RoboDK station: InvertedRobot003.rdk

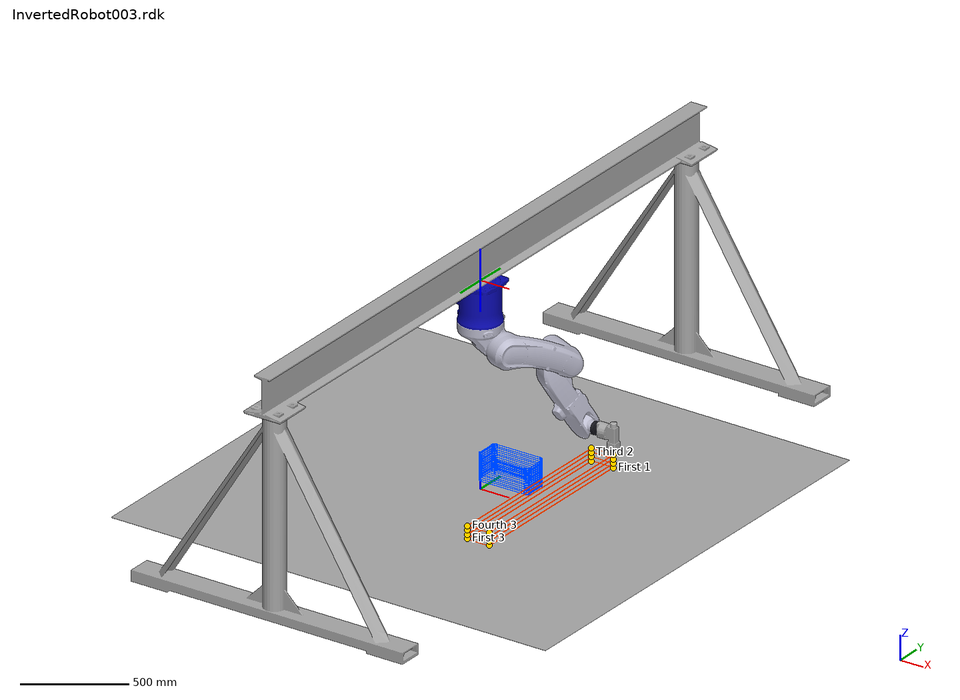
[picture v0: the station drawn from its stored meshes, robots at their saved joint values, targets as dots, program paths as lines]
Station InvertedRobot003 (saved by RoboDK 5.5.4). Poses are relative to the parent item; angles as X-Y-Z fixed-axis rotations.
Station parameters (name, value as stored): TAGS, ['Additive Manufacturing', 'Additive manufacturing']
  - frame Denso 1 at (0, 0, 1066.8) mm, rotated rx -180 ry 0 rz 0 deg
    - robot Denso VS-6577G-B: 6 axes, payload 7 kg, reach 854 mm, repeatability 0.03 mm, weight 36 kg
        modified DH rows (alpha deg, a mm, theta deg, d mm): 0, 0, 0, 335; -90, 75, -90, 0; 0, 365, -90, 0; -90, 90, 0, 405; 90, 0, 0, 0; -90, 0, 0, 80
        joint limits [-170, -100, -119, -190, -120, -360] to [170, 135, 169, 190, 120, 360]; home [0, 0, 90, 0, 0, 0]; saved at [-64.134, 67.115, -35.034, 67.667, 76.602, -29.424]
      - tool nozzle, TCP at (110, 0, 80) mm, rotated rx 0 ry 90 rz 0 deg, size 158.8 x 76.2 x 114.9 mm, geometry from nozzle.STEP
  - frame Ref001 at (0, 0, 0) mm
    - object Part at (0, 0, 0) mm, size 120 x 120 x 160 mm, geometry from part.sld
    - target First 1 (Cartesian target) at (400, 495, 22.23) mm, rotated rx 180 ry 0 rz 180 deg; joints [-64.134, 50.356, -9.939, 69.739, 73.569, -37.461] of Denso VS-6577G-B
    - target First 2 (Cartesian target) at (278, 495, 22.23) mm, rotated rx 180 ry 0 rz 180 deg; joints [-76.592, 55.531, -24.311, 78.477, 83.097, -30.522] of Denso VS-6577G-B
    - target First 3 (Cartesian target) at (278, -500, 22.23) mm, rotated rx 180 ry 0 rz 180 deg; joints [76.721, 17.283, 48.008, -84.366, 77.956, 64.696] of Denso VS-6577G-B
    - target First 4 (Cartesian target) at (400, -500, 22.23) mm, rotated rx 180 ry 0 rz 180 deg; joints [64.359, 49.428, -7.705, -70.29, 73.262, 38.795] of Denso VS-6577G-B
    - target Second 1 (Cartesian target) at (400, 495, 44.45) mm, rotated rx 180 ry 0 rz -180 deg; joints [-64.134, 57.09, -20.57, 68.712, 74.952, -33.676] of Denso VS-6577G-B
    - target Second 2 (Cartesian target) at (278, 495, 44.45) mm, rotated rx 180 ry 0 rz -180 deg; joints [-76.592, 60.643, -31.914, 78.193, 83.601, -28.066] of Denso VS-6577G-B
    - target Second 3 (Cartesian target) at (278, -500, 44.45) mm, rotated rx 180 ry 0 rz -180 deg; joints [76.721, 60.327, -30.755, -78.401, 83.491, 28.91] of Denso VS-6577G-B
    - target Second 4 (Cartesian target) at (400, -500, 44.45) mm, rotated rx 180 ry 0 rz -180 deg; joints [64.359, 56.542, -19.05, -69.151, 74.729, 34.667] of Denso VS-6577G-B
    - target Third 1 (Cartesian target) at (400, 495, 66.67) mm, rotated rx 180 ry 0 rz -180 deg; joints [-64.134, 62.433, -28.479, 68.091, 75.897, -31.211] of Denso VS-6577G-B
    - target Third 2 (Cartesian target) at (278, 495, 66.67) mm, rotated rx 180 ry 0 rz 180 deg; joints [-76.592, 65.197, -38.359, 77.992, 83.991, -26.205] of Denso VS-6577G-B
    - target Third 3 (Cartesian target) at (278, -500, 66.67) mm, rotated rx 180 ry 0 rz 180 deg; joints [76.721, 64.945, -37.316, -78.19, 83.885, 26.996] of Denso VS-6577G-B
    - target Third 4 (Cartesian target) at (400, -500, 66.67) mm, rotated rx 180 ry 0 rz 180 deg; joints [64.359, 62.027, -27.223, -68.489, 75.701, 32.074] of Denso VS-6577G-B
    - target Fourth 1 (Cartesian target) at (400, 495, 88.9) mm, rotated rx 180 ry 0 rz 180 deg; joints [-64.134, 67.115, -35.034, 67.667, 76.602, -29.424] of Denso VS-6577G-B
    - target Fourth 2 (Cartesian target) at (278, 495, 88.9) mm, rotated rx 180 ry 0 rz 180 deg; joints [-76.592, 69.405, -44.036, 77.844, 84.298, -24.761] of Denso VS-6577G-B
    - target Fourth 3 (Cartesian target) at (278, -500, 88.9) mm, rotated rx 180 ry 0 rz 180 deg; joints [76.721, 69.194, -43.068, -78.037, 84.195, 25.517] of Denso VS-6577G-B
    - target Fourth 4 (Cartesian target) at (400, -500, 88.9) mm, rotated rx 180 ry 0 rz 180 deg; joints [64.359, 66.785, -33.922, -68.041, 76.419, 30.216] of Denso VS-6577G-B
  - machining project Print3D settings: C:/Users/silverBlacK/OneDrive - University of Idaho/Research/RoboticsResearch/WallSection.gcode | rotZ(0) | rotX(0)*rotY(0) | rotZ(0)
  - program Print3D (17608 instructions, listed below)
  - frame Frame 4 at (0, 0, 1066.8) mm
    - object GantryAssembly at (0, 0, 0) mm, size 1524 x 3505.2 x 1270 mm, geometry from GantryAssembly.STEP
  - frame GarageFloor at (0, 0, 0) mm
    - object GarageFloor at (0, 0, 0) mm, size 2438.4 x 2438.4 x 2.5 mm, geometry from GarageFloor.STEP
  - program Prog4 (22 instructions, listed below)
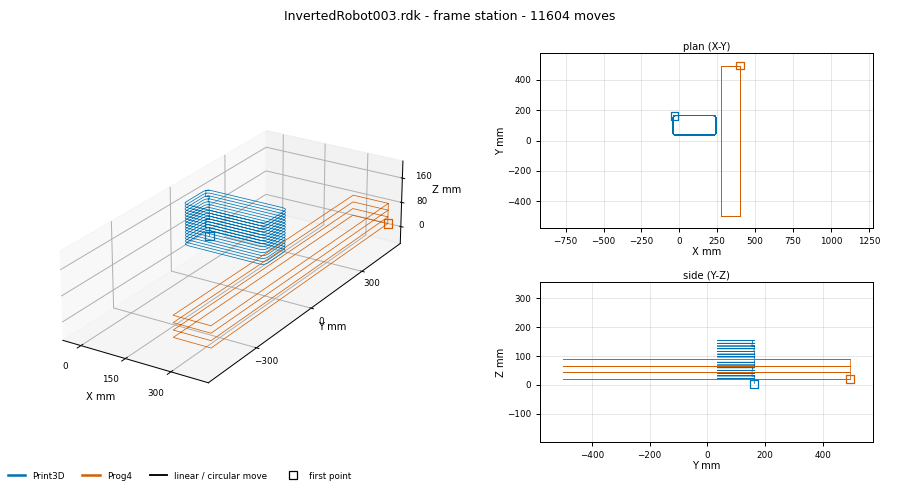
[picture p0: tool path of InvertedRobot003.rdk in frame station, 11604 of 11604 moves have a stored position in this frame; points joined in program order, loops and branches not executed]

--- program Print3D (robot Denso VS-6577G-B) ---
  Smooth(1)
  Call M_RunCode(107)
  Call M_RunCode(104)
  Set speed (83.3 mm/s)
  Set speed (1000.0 mm/s)
  Set Ref.: Ref001
  Set Tool: nozzle
  Show nozzle
  MoveJ 1 to (-31.64, 163.21, 5) mm, rotated rx -180 ry 0 rz 180 deg; joints [-139.581, 53.249, -56.919, 139.523, 87.207, 2.381]
  MoveL 2 to (-31.64, 163.21, 5) mm, rotated rx -180 ry 0 rz 180 deg; joints [-139.581, 53.249, -56.919, 139.523, 87.207, 2.381]
  Call Extruder(-1)
  MoveL 3 to (-31.64, 163.21, 5) mm, rotated rx -180 ry 0 rz 180 deg; joints [-139.581, 53.249, -56.919, 139.523, 87.207, 2.381]
  Call M_RunCode(109)
  Call M_RunCode(82)
  Call Extruder(0.00000)
  Set speed (130.0 mm/s)
  MoveL 4 to (-31.64, 163.21, 22.22) mm, rotated rx 180 ry 0 rz -180 deg; joints [-139.581, 55.977, -61.099, 139.468, 86.103, 3.326]
  Call Extruder(-2.00000)
  Set speed (40.0 mm/s)
  MoveL 5 to (-31.64, 163.21, 22.22) mm, rotated rx 180 ry 0 rz -180 deg; joints [-139.581, 55.977, -61.099, 139.468, 86.103, 3.326]
  Call Extruder(0.00000)
  Set speed (130.0 mm/s)
  MoveL 6 to (-31.64, 163.21, 22.22) mm, rotated rx 180 ry 0 rz -180 deg; joints [-139.581, 55.977, -61.099, 139.468, 86.103, 3.326]
  Call Extruder(2.00000)
  Set speed (40.0 mm/s)
  MoveL 7 to (-31.64, 163.21, 22.22) mm, rotated rx 180 ry 0 rz -180 deg; joints [-139.581, 55.977, -61.099, 139.468, 86.103, 3.326]
  Set speed (30.0 mm/s)
  MoveL 8 to (-31.64, 163.21, 22.22) mm, rotated rx 180 ry 0 rz -180 deg; joints [-139.581, 55.977, -61.099, 139.468, 86.103, 3.326]
  Call Extruder(2.38024)
  MoveL 9 to (-31.93, 163.09, 22.22) mm, rotated rx -180 ry 0 rz 180 deg; joints [-139.645, 55.984, -61.089, 139.532, 86.112, 3.311]
  MoveL 10 to (-31.93, 163.09, 22.22) mm, rotated rx -180 ry 0 rz 180 deg; joints [-139.645, 55.984, -61.089, 139.532, 86.112, 3.311]
  Call Extruder(2.76227)
  MoveL 11 to (-32.22, 162.97, 22.23) mm, rotated rx -180 ry 0 rz -180 deg; joints [-139.709, 55.991, -61.079, 139.597, 86.121, 3.295]
  MoveL 12 to (-32.22, 162.97, 22.23) mm, rotated rx -180 ry 0 rz -180 deg; joints [-139.709, 55.991, -61.079, 139.597, 86.121, 3.295]
  Call Extruder(3.11872)
  MoveL 13 to (-32.49, 162.85, 22.22) mm, rotated rx 180 ry 0 rz 180 deg; joints [-139.768, 55.998, -61.07, 139.657, 86.13, 3.281]
  MoveL 14 to (-32.49, 162.85, 22.22) mm, rotated rx 180 ry 0 rz 180 deg; joints [-139.768, 55.998, -61.07, 139.657, 86.13, 3.281]
  Call Extruder(3.44932)
  MoveL 15 to (-32.74, 162.74, 22.22) mm, rotated rx -180 ry 0 rz 180 deg; joints [-139.823, 56.004, -61.061, 139.713, 86.138, 3.268]
  MoveL 16 to (-32.74, 162.74, 22.22) mm, rotated rx -180 ry 0 rz 180 deg; joints [-139.823, 56.004, -61.061, 139.713, 86.138, 3.268]
  Call Extruder(3.78134)
  MoveL 17 to (-32.99, 162.64, 22.22) mm, rotated rx 180 ry 0 rz -180 deg; joints [-139.878, 56.01, -61.053, 139.769, 86.146, 3.255]
  MoveL 18 to (-32.99, 162.64, 22.22) mm, rotated rx 180 ry 0 rz -180 deg; joints [-139.878, 56.01, -61.053, 139.769, 86.146, 3.255]
  Call Extruder(4.21321)
  MoveL 19 to (-33.29, 162.46, 22.22) mm, rotated rx -180 ry 0 rz 180 deg; joints [-139.953, 56.016, -61.044, 139.844, 86.152, 3.24]
  MoveL 20 to (-33.29, 162.46, 22.22) mm, rotated rx -180 ry 0 rz 180 deg; joints [-139.953, 56.016, -61.044, 139.844, 86.152, 3.24]
  Call Extruder(4.64692)
  MoveL 21 to (-33.6, 162.29, 22.22) mm, rotated rx 180 ry 0 rz 180 deg; joints [-140.028, 56.022, -61.036, 139.92, 86.159, 3.226]
  MoveL 22 to (-33.6, 162.29, 22.22) mm, rotated rx 180 ry 0 rz 180 deg; joints [-140.028, 56.022, -61.036, 139.92, 86.159, 3.226]
  Call Extruder(5.08247)
  MoveL 23 to (-33.9, 162.11, 22.22) mm, rotated rx -180 ry 0 rz 180 deg; joints [-140.103, 56.027, -61.028, 139.995, 86.166, 3.212]
  MoveL 24 to (-33.9, 162.11, 22.22) mm, rotated rx -180 ry 0 rz 180 deg; joints [-140.103, 56.027, -61.028, 139.995, 86.166, 3.212]
  Call Extruder(5.51986)
  MoveL 25 to (-34.21, 161.93, 22.22) mm, rotated rx -180 ry 0 rz -180 deg; joints [-140.178, 56.033, -61.019, 140.071, 86.173, 3.198]
  MoveL 26 to (-34.21, 161.93, 22.22) mm, rotated rx -180 ry 0 rz -180 deg; joints [-140.178, 56.033, -61.019, 140.071, 86.173, 3.198]
  Call Extruder(5.89660)
  MoveL 27 to (-34.45, 161.76, 22.23) mm, rotated rx -180 ry 0 rz 180 deg; joints [-140.244, 56.037, -61.014, 140.137, 86.176, 3.187]
  MoveL 28 to (-34.45, 161.76, 22.23) mm, rotated rx -180 ry 0 rz 180 deg; joints [-140.244, 56.037, -61.014, 140.137, 86.176, 3.187]
  Call Extruder(6.59657)
  MoveL 29 to (-34.9, 161.43, 22.22) mm, rotated rx 180 ry 0 rz -180 deg; joints [-140.366, 56.044, -61.004, 140.261, 86.182, 3.169]
  MoveL 30 to (-34.9, 161.43, 22.22) mm, rotated rx 180 ry 0 rz -180 deg; joints [-140.366, 56.044, -61.004, 140.261, 86.182, 3.169]
  Call Extruder(7.29934)
  MoveL 31 to (-35.35, 161.1, 22.22) mm, rotated rx -180 ry 0 rz -180 deg; joints [-140.489, 56.051, -60.994, 140.384, 86.188, 3.15]
  Call Extruder(9.03811)
  MoveL 32 to (-36.39, 160.19, 22.22) mm, rotated rx -180 ry 0 rz 180 deg; joints [-140.797, 56.062, -60.979, 140.693, 86.192, 3.112]
  Call Extruder(10.77694)
  MoveL 33 to (-37.3, 159.15, 22.22) mm, rotated rx -180 ry 0 rz -180 deg; joints [-141.109, 56.064, -60.975, 141.006, 86.18, 3.087]
  Call Extruder(11.12832)
  MoveL 34 to (-37.47, 158.93, 22.22) mm, rotated rx -180 ry 0 rz -180 deg; joints [-141.172, 56.064, -60.976, 141.069, 86.175, 3.084]
  MoveL 35 to (-37.47, 158.93, 22.22) mm, rotated rx -180 ry 0 rz -180 deg; joints [-141.172, 56.064, -60.976, 141.069, 86.175, 3.084]
  Call Extruder(11.82828)
  MoveL 36 to (-37.8, 158.48, 22.22) mm, rotated rx 180 ry 0 rz 180 deg; joints [-141.298, 56.062, -60.978, 141.195, 86.166, 3.078]
  MoveL 37 to (-37.8, 158.48, 22.22) mm, rotated rx 180 ry 0 rz 180 deg; joints [-141.298, 56.062, -60.978, 141.195, 86.166, 3.078]
  Call Extruder(12.52544)
  MoveL 38 to (-38.12, 158.03, 22.22) mm, rotated rx 180 ry 0 rz 180 deg; joints [-141.424, 56.061, -60.979, 141.321, 86.157, 3.071]
  MoveL 39 to (-38.12, 158.03, 22.22) mm, rotated rx 180 ry 0 rz 180 deg; joints [-141.424, 56.061, -60.979, 141.321, 86.157, 3.071]
  Call Extruder(12.77229)
  MoveL 40 to (-38.22, 157.85, 22.22) mm, rotated rx -180 ry 0 rz 180 deg; joints [-141.468, 56.06, -60.981, 141.365, 86.152, 3.071]
  MoveL 41 to (-38.22, 157.85, 22.22) mm, rotated rx -180 ry 0 rz 180 deg; joints [-141.468, 56.06, -60.981, 141.365, 86.152, 3.071]
  Call Extruder(13.20785)
  MoveL 42 to (-38.4, 157.55, 22.22) mm, rotated rx 180 ry 0 rz -180 deg; joints [-141.547, 56.057, -60.985, 141.443, 86.143, 3.069]
  MoveL 43 to (-38.4, 157.55, 22.22) mm, rotated rx 180 ry 0 rz -180 deg; joints [-141.547, 56.057, -60.985, 141.443, 86.143, 3.069]
  Call Extruder(13.64157)
  MoveL 44 to (-38.57, 157.25, 22.22) mm, rotated rx 180 ry 0 rz 180 deg; joints [-141.625, 56.055, -60.989, 141.522, 86.134, 3.068]
  MoveL 45 to (-38.57, 157.25, 22.22) mm, rotated rx 180 ry 0 rz 180 deg; joints [-141.625, 56.055, -60.989, 141.522, 86.134, 3.068]
  Call Extruder(14.07344)
  MoveL 46 to (-38.75, 156.94, 22.23) mm, rotated rx 180 ry 0 rz 180 deg; joints [-141.704, 56.052, -60.992, 141.6, 86.125, 3.066]
  MoveL 47 to (-38.75, 156.94, 22.23) mm, rotated rx 180 ry 0 rz 180 deg; joints [-141.704, 56.052, -60.992, 141.6, 86.125, 3.066]
  Call Extruder(14.45383)
  MoveL 48 to (-38.89, 156.67, 22.22) mm, rotated rx -180 ry 0 rz -180 deg; joints [-141.773, 56.049, -60.996, 141.669, 86.115, 3.066]
  MoveL 49 to (-38.89, 156.67, 22.22) mm, rotated rx -180 ry 0 rz -180 deg; joints [-141.773, 56.049, -60.996, 141.669, 86.115, 3.066]
  Call Extruder(14.78446)
  MoveL 50 to (-39, 156.42, 22.22) mm, rotated rx -180 ry 0 rz 180 deg; joints [-141.832, 56.046, -61.001, 141.728, 86.106, 3.067]
  MoveL 51 to (-39, 156.42, 22.22) mm, rotated rx -180 ry 0 rz 180 deg; joints [-141.832, 56.046, -61.001, 141.728, 86.106, 3.067]
  Call Extruder(15.11366)
  MoveL 52 to (-39.1, 156.17, 22.22) mm, rotated rx -180 ry 0 rz -180 deg; joints [-141.891, 56.042, -61.006, 141.787, 86.096, 3.068]
  MoveL 53 to (-39.1, 156.17, 22.22) mm, rotated rx -180 ry 0 rz -180 deg; joints [-141.891, 56.042, -61.006, 141.787, 86.096, 3.068]
  Call Extruder(15.49565)
  MoveL 54 to (-39.22, 155.87, 22.23) mm, rotated rx -180 ry 0 rz 180 deg; joints [-141.96, 56.038, -61.012, 141.855, 86.084, 3.07]
  MoveL 55 to (-39.22, 155.87, 22.23) mm, rotated rx -180 ry 0 rz 180 deg; joints [-141.96, 56.038, -61.012, 141.855, 86.084, 3.07]
  Call Extruder(15.87585)
  MoveL 56 to (-39.35, 155.58, 22.23) mm, rotated rx 180 ry 0 rz 180 deg; joints [-142.029, 56.034, -61.018, 141.924, 86.073, 3.071]
  MoveL 57 to (-39.35, 155.58, 22.23) mm, rotated rx 180 ry 0 rz 180 deg; joints [-142.029, 56.034, -61.018, 141.924, 86.073, 3.071]
  Call Extruder(16.18353)
  MoveL 58 to (-39.44, 155.34, 22.22) mm, rotated rx 180 ry 0 rz 180 deg; joints [-142.085, 56.03, -61.024, 141.979, 86.063, 3.073]
  MoveL 59 to (-39.44, 155.34, 22.22) mm, rotated rx 180 ry 0 rz 180 deg; joints [-142.085, 56.03, -61.024, 141.979, 86.063, 3.073]
  Call Extruder(16.41988)
  MoveL 60 to (-39.5, 155.15, 22.22) mm, rotated rx -180 ry 0 rz 180 deg; joints [-142.127, 56.027, -61.028, 142.021, 86.054, 3.075]
  MoveL 61 to (-39.5, 155.15, 22.22) mm, rotated rx -180 ry 0 rz 180 deg; joints [-142.127, 56.027, -61.028, 142.021, 86.054, 3.075]
  Call Extruder(16.65518)
  MoveL 62 to (-39.56, 154.97, 22.22) mm, rotated rx -180 ry 0 rz 180 deg; joints [-142.169, 56.024, -61.033, 142.063, 86.045, 3.077]
  MoveL 63 to (-39.56, 154.97, 22.22) mm, rotated rx -180 ry 0 rz 180 deg; joints [-142.169, 56.024, -61.033, 142.063, 86.045, 3.077]
  Call Extruder(16.88943)
  MoveL 64 to (-39.62, 154.78, 22.22) mm, rotated rx 180 ry 0 rz 180 deg; joints [-142.212, 56.02, -61.038, 142.105, 86.037, 3.079]
  MoveL 65 to (-39.62, 154.78, 22.22) mm, rotated rx 180 ry 0 rz 180 deg; joints [-142.212, 56.02, -61.038, 142.105, 86.037, 3.079]
  Call Extruder(17.12262)
  MoveL 66 to (-39.68, 154.59, 22.22) mm, rotated rx -180 ry 0 rz -180 deg; joints [-142.254, 56.017, -61.042, 142.147, 86.028, 3.081]
  MoveL 67 to (-39.68, 154.59, 22.22) mm, rotated rx -180 ry 0 rz -180 deg; joints [-142.254, 56.017, -61.042, 142.147, 86.028, 3.081]
  Call Extruder(17.37548)
  MoveL 68 to (-39.75, 154.38, 22.22) mm, rotated rx -180 ry 0 rz 180 deg; joints [-142.3, 56.013, -61.048, 142.193, 86.019, 3.084]
  MoveL 69 to (-39.75, 154.38, 22.22) mm, rotated rx -180 ry 0 rz 180 deg; joints [-142.3, 56.013, -61.048, 142.193, 86.019, 3.084]
  Call Extruder(17.64775)
  MoveL 70 to (-39.81, 154.16, 22.22) mm, rotated rx 180 ry 0 rz 180 deg; joints [-142.35, 56.009, -61.053, 142.242, 86.008, 3.086]
  MoveL 71 to (-39.81, 154.16, 22.22) mm, rotated rx 180 ry 0 rz 180 deg; joints [-142.35, 56.009, -61.053, 142.242, 86.008, 3.086]
  Call Extruder(17.91868)
  MoveL 72 to (-39.88, 153.94, 22.22) mm, rotated rx 180 ry 0 rz -180 deg; joints [-142.399, 56.005, -61.059, 142.291, 85.998, 3.089]
  MoveL 73 to (-39.88, 153.94, 22.22) mm, rotated rx 180 ry 0 rz -180 deg; joints [-142.399, 56.005, -61.059, 142.291, 85.998, 3.089]
  Call Extruder(18.18828)
  MoveL 74 to (-39.95, 153.71, 22.23) mm, rotated rx -180 ry 0 rz -180 deg; joints [-142.449, 56.001, -61.065, 142.34, 85.987, 3.091]
  MoveL 75 to (-39.95, 153.71, 22.23) mm, rotated rx -180 ry 0 rz -180 deg; joints [-142.449, 56.001, -61.065, 142.34, 85.987, 3.091]
  Call Extruder(18.45654)
  MoveL 76 to (-40.02, 153.49, 22.22) mm, rotated rx -180 ry 0 rz -180 deg; joints [-142.498, 55.997, -61.071, 142.39, 85.977, 3.094]
  MoveL 77 to (-40.02, 153.49, 22.22) mm, rotated rx -180 ry 0 rz -180 deg; joints [-142.498, 55.997, -61.071, 142.39, 85.977, 3.094]
  Call Extruder(18.69554)
  MoveL 78 to (-40.06, 153.28, 22.22) mm, rotated rx -180 ry 0 rz 180 deg; joints [-142.541, 55.993, -61.077, 142.432, 85.966, 3.097]
  MoveL 79 to (-40.06, 153.28, 22.22) mm, rotated rx -180 ry 0 rz 180 deg; joints [-142.541, 55.993, -61.077, 142.432, 85.966, 3.097]
  Call Extruder(18.93348)
  MoveL 80 to (-40.11, 153.08, 22.22) mm, rotated rx 180 ry 0 rz 180 deg; joints [-142.584, 55.988, -61.083, 142.475, 85.955, 3.101]
  MoveL 81 to (-40.11, 153.08, 22.22) mm, rotated rx 180 ry 0 rz 180 deg; joints [-142.584, 55.988, -61.083, 142.475, 85.955, 3.101]
  Call Extruder(19.17035)
  MoveL 82 to (-40.15, 152.88, 22.22) mm, rotated rx -180 ry 0 rz 180 deg; joints [-142.627, 55.984, -61.089, 142.517, 85.945, 3.104]
  MoveL 83 to (-40.15, 152.88, 22.22) mm, rotated rx -180 ry 0 rz 180 deg; joints [-142.627, 55.984, -61.089, 142.517, 85.945, 3.104]
  Call Extruder(19.40615)
  MoveL 84 to (-40.2, 152.67, 22.22) mm, rotated rx -180 ry 0 rz 180 deg; joints [-142.671, 55.979, -61.096, 142.56, 85.934, 3.108]
  MoveL 85 to (-40.2, 152.67, 22.22) mm, rotated rx -180 ry 0 rz 180 deg; joints [-142.671, 55.979, -61.096, 142.56, 85.934, 3.108]
  Call Extruder(19.66605)
  MoveL 86 to (-40.24, 152.44, 22.22) mm, rotated rx 180 ry 0 rz 180 deg; joints [-142.718, 55.974, -61.103, 142.607, 85.922, 3.112]
  MoveL 87 to (-40.24, 152.44, 22.22) mm, rotated rx 180 ry 0 rz 180 deg; joints [-142.718, 55.974, -61.103, 142.607, 85.922, 3.112]
  Call Extruder(19.94972)
  MoveL 88 to (-40.29, 152.2, 22.23) mm, rotated rx -180 ry 0 rz -180 deg; joints [-142.77, 55.969, -61.11, 142.659, 85.908, 3.116]
  MoveL 89 to (-40.29, 152.2, 22.23) mm, rotated rx -180 ry 0 rz -180 deg; joints [-142.77, 55.969, -61.11, 142.659, 85.908, 3.116]
  Call Extruder(20.23193)
  MoveL 90 to (-40.34, 151.95, 22.22) mm, rotated rx -180 ry 0 rz -180 deg; joints [-142.822, 55.963, -61.118, 142.71, 85.895, 3.12]
  MoveL 91 to (-40.34, 151.95, 22.22) mm, rotated rx -180 ry 0 rz -180 deg; joints [-142.822, 55.963, -61.118, 142.71, 85.895, 3.12]
  Call Extruder(20.51271)
  MoveL 92 to (-40.39, 151.7, 22.22) mm, rotated rx 180 ry 0 rz 180 deg; joints [-142.874, 55.958, -61.126, 142.762, 85.882, 3.125]
  MoveL 93 to (-40.39, 151.7, 22.22) mm, rotated rx 180 ry 0 rz 180 deg; joints [-142.874, 55.958, -61.126, 142.762, 85.882, 3.125]
  Call Extruder(20.79205)
  MoveL 94 to (-40.44, 151.45, 22.23) mm, rotated rx 180 ry 0 rz 180 deg; joints [-142.926, 55.952, -61.133, 142.813, 85.868, 3.129]
  MoveL 95 to (-40.44, 151.45, 22.23) mm, rotated rx 180 ry 0 rz 180 deg; joints [-142.926, 55.952, -61.133, 142.813, 85.868, 3.129]
  Call Extruder(21.06994)
  MoveL 96 to (-40.49, 151.2, 22.23) mm, rotated rx -180 ry 0 rz 180 deg; joints [-142.978, 55.947, -61.141, 142.865, 85.855, 3.133]
  MoveL 97 to (-40.49, 151.2, 22.23) mm, rotated rx -180 ry 0 rz 180 deg; joints [-142.978, 55.947, -61.141, 142.865, 85.855, 3.133]
  Call Extruder(21.34639)
  MoveL 98 to (-40.54, 150.95, 22.23) mm, rotated rx 180 ry 0 rz 180 deg; joints [-143.031, 55.941, -61.149, 142.917, 85.842, 3.137]
  MoveL 99 to (-40.54, 150.95, 22.23) mm, rotated rx 180 ry 0 rz 180 deg; joints [-143.031, 55.941, -61.149, 142.917, 85.842, 3.137]
  Call Extruder(21.65140)
  MoveL 100 to (-40.59, 150.67, 22.22) mm, rotated rx -180 ry 0 rz -180 deg; joints [-143.088, 55.935, -61.158, 142.973, 85.826, 3.142]
  MoveL 101 to (-40.59, 150.67, 22.22) mm, rotated rx -180 ry 0 rz -180 deg; joints [-143.088, 55.935, -61.158, 142.973, 85.826, 3.142]
  Call Extruder(21.98479)
  MoveL 102 to (-40.64, 150.37, 22.22) mm, rotated rx 180 ry 0 rz -180 deg; joints [-143.15, 55.928, -61.168, 143.035, 85.809, 3.148]
  MoveL 103 to (-40.64, 150.37, 22.22) mm, rotated rx 180 ry 0 rz -180 deg; joints [-143.15, 55.928, -61.168, 143.035, 85.809, 3.148]
  Call Extruder(22.31647)
  MoveL 104 to (-40.69, 150.06, 22.22) mm, rotated rx 180 ry 0 rz 180 deg; joints [-143.213, 55.921, -61.178, 143.097, 85.792, 3.154]
  MoveL 105 to (-40.69, 150.06, 22.22) mm, rotated rx 180 ry 0 rz 180 deg; joints [-143.213, 55.921, -61.178, 143.097, 85.792, 3.154]
  Call Extruder(22.64643)
  MoveL 106 to (-40.74, 149.76, 22.22) mm, rotated rx -180 ry 0 rz -180 deg; joints [-143.276, 55.913, -61.188, 143.159, 85.775, 3.16]
  MoveL 107 to (-40.74, 149.76, 22.22) mm, rotated rx -180 ry 0 rz -180 deg; joints [-143.276, 55.913, -61.188, 143.159, 85.775, 3.16]
  Call Extruder(22.97467)
  MoveL 108 to (-40.78, 149.45, 22.22) mm, rotated rx 180 ry 0 rz 180 deg; joints [-143.338, 55.906, -61.198, 143.221, 85.758, 3.165]
  MoveL 109 to (-40.78, 149.45, 22.22) mm, rotated rx 180 ry 0 rz 180 deg; joints [-143.338, 55.906, -61.198, 143.221, 85.758, 3.165]
  Call Extruder(23.30119)
  MoveL 110 to (-40.83, 149.14, 22.22) mm, rotated rx -180 ry 0 rz 180 deg; joints [-143.401, 55.899, -61.207, 143.283, 85.74, 3.171]
  MoveL 111 to (-40.83, 149.14, 22.22) mm, rotated rx -180 ry 0 rz 180 deg; joints [-143.401, 55.899, -61.207, 143.283, 85.74, 3.171]
  Call Extruder(23.66827)
  MoveL 112 to (-40.88, 148.8, 22.22) mm, rotated rx -180 ry 0 rz 180 deg; joints [-143.471, 55.891, -61.219, 143.353, 85.72, 3.178]
  MoveL 113 to (-40.88, 148.8, 22.22) mm, rotated rx -180 ry 0 rz 180 deg; joints [-143.471, 55.891, -61.219, 143.353, 85.72, 3.178]
  Call Extruder(24.07571)
  MoveL 114 to (-40.93, 148.41, 22.22) mm, rotated rx 180 ry 0 rz 180 deg; joints [-143.549, 55.881, -61.232, 143.429, 85.698, 3.186]
  MoveL 115 to (-40.93, 148.41, 22.22) mm, rotated rx 180 ry 0 rz 180 deg; joints [-143.549, 55.881, -61.232, 143.429, 85.698, 3.186]
  Call Extruder(24.48110)
  MoveL 116 to (-40.97, 148.02, 22.22) mm, rotated rx -180 ry 0 rz -180 deg; joints [-143.627, 55.871, -61.246, 143.506, 85.675, 3.193]
  MoveL 117 to (-40.97, 148.02, 22.22) mm, rotated rx -180 ry 0 rz -180 deg; joints [-143.627, 55.871, -61.246, 143.506, 85.675, 3.193]
  Call Extruder(24.88445)
  MoveL 118 to (-41.02, 147.63, 22.22) mm, rotated rx -180 ry 0 rz -180 deg; joints [-143.705, 55.861, -61.259, 143.583, 85.652, 3.201]
  MoveL 119 to (-41.02, 147.63, 22.22) mm, rotated rx -180 ry 0 rz -180 deg; joints [-143.705, 55.861, -61.259, 143.583, 85.652, 3.201]
  Call Extruder(25.28574)
  MoveL 120 to (-41.06, 147.25, 22.22) mm, rotated rx 180 ry 0 rz 180 deg; joints [-143.783, 55.852, -61.272, 143.66, 85.629, 3.209]
  MoveL 121 to (-41.06, 147.25, 22.22) mm, rotated rx 180 ry 0 rz 180 deg; joints [-143.783, 55.852, -61.272, 143.66, 85.629, 3.209]
  Call Extruder(25.89062)
  MoveL 122 to (-41.11, 146.66, 22.22) mm, rotated rx 180 ry 0 rz -180 deg; joints [-143.899, 55.836, -61.293, 143.775, 85.593, 3.222]
  MoveL 123 to (-41.11, 146.66, 22.22) mm, rotated rx 180 ry 0 rz -180 deg; joints [-143.899, 55.836, -61.293, 143.775, 85.593, 3.222]
  Call Extruder(26.49235)
  MoveL 124 to (-41.16, 146.07, 22.22) mm, rotated rx -180 ry 0 rz -180 deg; joints [-144.015, 55.82, -61.315, 143.889, 85.557, 3.235]
  MoveL 125 to (-41.16, 146.07, 22.22) mm, rotated rx -180 ry 0 rz -180 deg; joints [-144.015, 55.82, -61.315, 143.889, 85.557, 3.235]
  Call Extruder(27.09093)
  MoveL 126 to (-41.2, 145.48, 22.22) mm, rotated rx 180 ry 0 rz 180 deg; joints [-144.131, 55.805, -61.336, 144.004, 85.52, 3.247]
  MoveL 127 to (-41.2, 145.48, 22.22) mm, rotated rx 180 ry 0 rz 180 deg; joints [-144.131, 55.805, -61.336, 144.004, 85.52, 3.247]
  Call Extruder(28.26271)
  MoveL 128 to (-41.25, 144.32, 22.22) mm, rotated rx 180 ry 0 rz 180 deg; joints [-144.355, 55.772, -61.379, 144.225, 85.446, 3.274]
  MoveL 129 to (-41.25, 144.32, 22.22) mm, rotated rx 180 ry 0 rz 180 deg; joints [-144.355, 55.772, -61.379, 144.225, 85.446, 3.274]
  Call Extruder(29.72057)
  MoveL 130 to (-41.29, 142.86, 22.22) mm, rotated rx -180 ry 0 rz 180 deg; joints [-144.635, 55.731, -61.434, 144.501, 85.351, 3.308]
  Call Extruder(115.61408)
  MoveL 131 to (-41.29, 57.14, 22.22) mm, rotated rx -180 ry 0 rz 180 deg; joints [-164.153, 53.6, -63.687, 163.917, 80.3, 2.781]
  Call Extruder(116.48916)
  MoveL 132 to (-41.27, 56.26, 22.22) mm, rotated rx -180 ry 0 rz 180 deg; joints [-164.382, 53.584, -63.7, 164.148, 80.261, 2.75]
  MoveL 133 to (-41.27, 56.26, 22.22) mm, rotated rx -180 ry 0 rz 180 deg; joints [-164.382, 53.584, -63.7, 164.148, 80.261, 2.75]
  Call Extruder(117.66094)
  MoveL 134 to (-41.22, 55.1, 22.22) mm, rotated rx 180 ry 0 rz 180 deg; joints [-164.686, 53.562, -63.719, 164.454, 80.207, 2.709]
  MoveL 135 to (-41.22, 55.1, 22.22) mm, rotated rx 180 ry 0 rz 180 deg; joints [-164.686, 53.562, -63.719, 164.454, 80.207, 2.709]
  Call Extruder(118.54904)
  MoveL 136 to (-41.18, 54.23, 22.23) mm, rotated rx 180 ry 0 rz -180 deg; joints [-164.915, 53.545, -63.733, 164.685, 80.166, 2.678]
  MoveL 137 to (-41.18, 54.23, 22.23) mm, rotated rx 180 ry 0 rz -180 deg; joints [-164.915, 53.545, -63.733, 164.685, 80.166, 2.678]
  Call Extruder(119.15077)
  MoveL 138 to (-41.13, 53.64, 22.22) mm, rotated rx 180 ry 0 rz 180 deg; joints [-165.068, 53.532, -63.743, 164.839, 80.137, 2.657]
  MoveL 139 to (-41.13, 53.64, 22.22) mm, rotated rx 180 ry 0 rz 180 deg; joints [-165.068, 53.532, -63.743, 164.839, 80.137, 2.657]
  Call Extruder(119.75565)
  MoveL 140 to (-41.09, 53.05, 22.22) mm, rotated rx -180 ry 0 rz 180 deg; joints [-165.222, 53.52, -63.754, 164.994, 80.109, 2.637]
  MoveL 141 to (-41.09, 53.05, 22.22) mm, rotated rx -180 ry 0 rz 180 deg; joints [-165.222, 53.52, -63.754, 164.994, 80.109, 2.637]
  Call Extruder(120.26021)
  MoveL 142 to (-41.04, 52.56, 22.22) mm, rotated rx -180 ry 0 rz -180 deg; joints [-165.349, 53.51, -63.762, 165.121, 80.084, 2.619]
  MoveL 143 to (-41.04, 52.56, 22.22) mm, rotated rx -180 ry 0 rz -180 deg; joints [-165.349, 53.51, -63.762, 165.121, 80.084, 2.619]
  Call Extruder(120.66355)
  MoveL 144 to (-40.99, 52.17, 22.22) mm, rotated rx -180 ry 0 rz 180 deg; joints [-165.449, 53.501, -63.77, 165.223, 80.064, 2.606]
  MoveL 145 to (-40.99, 52.17, 22.22) mm, rotated rx -180 ry 0 rz 180 deg; joints [-165.449, 53.501, -63.77, 165.223, 80.064, 2.606]
  Call Extruder(121.06894)
  MoveL 146 to (-40.95, 51.78, 22.22) mm, rotated rx -180 ry 0 rz 180 deg; joints [-165.549, 53.492, -63.777, 165.323, 80.044, 2.593]
  MoveL 147 to (-40.95, 51.78, 22.22) mm, rotated rx -180 ry 0 rz 180 deg; joints [-165.549, 53.492, -63.777, 165.323, 80.044, 2.593]
  Call Extruder(121.47639)
  MoveL 148 to (-40.9, 51.4, 22.22) mm, rotated rx 180 ry 0 rz 180 deg; joints [-165.65, 53.483, -63.784, 165.425, 80.024, 2.579]
  MoveL 149 to (-40.9, 51.4, 22.22) mm, rotated rx 180 ry 0 rz 180 deg; joints [-165.65, 53.483, -63.784, 165.425, 80.024, 2.579]
  Call Extruder(121.88588)
  MoveL 150 to (-40.86, 51.01, 22.23) mm, rotated rx 180 ry 0 rz -180 deg; joints [-165.751, 53.474, -63.791, 165.526, 80.004, 2.566]
  MoveL 151 to (-40.86, 51.01, 22.23) mm, rotated rx 180 ry 0 rz -180 deg; joints [-165.751, 53.474, -63.791, 165.526, 80.004, 2.566]
  Call Extruder(122.21240)
  MoveL 152 to (-40.81, 50.7, 22.22) mm, rotated rx 180 ry 0 rz -180 deg; joints [-165.829, 53.467, -63.798, 165.605, 79.987, 2.555]
  MoveL 153 to (-40.81, 50.7, 22.22) mm, rotated rx 180 ry 0 rz -180 deg; joints [-165.829, 53.467, -63.798, 165.605, 79.987, 2.555]
  Call Extruder(122.54064)
  MoveL 154 to (-40.76, 50.4, 22.22) mm, rotated rx -180 ry 0 rz -180 deg; joints [-165.908, 53.459, -63.804, 165.685, 79.97, 2.545]
  MoveL 155 to (-40.76, 50.4, 22.22) mm, rotated rx -180 ry 0 rz -180 deg; joints [-165.908, 53.459, -63.804, 165.685, 79.97, 2.545]
  Call Extruder(122.87060)
  MoveL 156 to (-40.71, 50.09, 22.22) mm, rotated rx 180 ry 0 rz 180 deg; joints [-165.987, 53.451, -63.81, 165.764, 79.953, 2.534]
  MoveL 157 to (-40.71, 50.09, 22.22) mm, rotated rx 180 ry 0 rz 180 deg; joints [-165.987, 53.451, -63.81, 165.764, 79.953, 2.534]
  Call Extruder(123.20228)
  MoveL 158 to (-40.66, 49.79, 22.22) mm, rotated rx -180 ry 0 rz -180 deg; joints [-166.066, 53.444, -63.816, 165.844, 79.936, 2.524]
  MoveL 159 to (-40.66, 49.79, 22.22) mm, rotated rx -180 ry 0 rz -180 deg; joints [-166.066, 53.444, -63.816, 165.844, 79.936, 2.524]
  Call Extruder(123.53568)
  MoveL 160 to (-40.61, 49.48, 22.22) mm, rotated rx -180 ry 0 rz 180 deg; joints [-166.145, 53.436, -63.823, 165.923, 79.919, 2.513]
  MoveL 161 to (-40.61, 49.48, 22.22) mm, rotated rx -180 ry 0 rz 180 deg; joints [-166.145, 53.436, -63.823, 165.923, 79.919, 2.513]
  Call Extruder(123.87079)
  MoveL 162 to (-40.57, 49.17, 22.22) mm, rotated rx -180 ry 0 rz -180 deg; joints [-166.224, 53.429, -63.829, 166.003, 79.902, 2.503]
  MoveL 163 to (-40.57, 49.17, 22.22) mm, rotated rx -180 ry 0 rz -180 deg; joints [-166.224, 53.429, -63.829, 166.003, 79.902, 2.503]
  Call Extruder(124.14680)
  MoveL 164 to (-40.52, 48.93, 22.22) mm, rotated rx 180 ry 0 rz -180 deg; joints [-166.288, 53.422, -63.834, 166.067, 79.888, 2.494]
  MoveL 165 to (-40.52, 48.93, 22.22) mm, rotated rx 180 ry 0 rz -180 deg; joints [-166.288, 53.422, -63.834, 166.067, 79.888, 2.494]
  Call Extruder(124.42424)
  MoveL 166 to (-40.47, 48.68, 22.22) mm, rotated rx -180 ry 0 rz 180 deg; joints [-166.352, 53.415, -63.84, 166.131, 79.873, 2.486]
  MoveL 167 to (-40.47, 48.68, 22.22) mm, rotated rx -180 ry 0 rz 180 deg; joints [-166.352, 53.415, -63.84, 166.131, 79.873, 2.486]
  Call Extruder(124.70312)
  MoveL 168 to (-40.42, 48.43, 22.22) mm, rotated rx -180 ry 0 rz -180 deg; joints [-166.416, 53.409, -63.845, 166.196, 79.859, 2.477]
  MoveL 169 to (-40.42, 48.43, 22.22) mm, rotated rx -180 ry 0 rz -180 deg; joints [-166.416, 53.409, -63.845, 166.196, 79.859, 2.477]
  Call Extruder(124.98344)
  MoveL 170 to (-40.37, 48.18, 22.22) mm, rotated rx -180 ry 0 rz -180 deg; joints [-166.479, 53.402, -63.851, 166.26, 79.844, 2.469]
  MoveL 171 to (-40.37, 48.18, 22.22) mm, rotated rx -180 ry 0 rz -180 deg; joints [-166.479, 53.402, -63.851, 166.26, 79.844, 2.469]
  Call Extruder(125.26519)
  MoveL 172 to (-40.32, 47.93, 22.22) mm, rotated rx 180 ry 0 rz -180 deg; joints [-166.544, 53.395, -63.856, 166.325, 79.829, 2.46]
  MoveL 173 to (-40.32, 47.93, 22.22) mm, rotated rx 180 ry 0 rz -180 deg; joints [-166.544, 53.395, -63.856, 166.325, 79.829, 2.46]
  Call Extruder(125.54838)
  MoveL 174 to (-40.27, 47.68, 22.23) mm, rotated rx -180 ry 0 rz 180 deg; joints [-166.608, 53.388, -63.861, 166.389, 79.815, 2.452]
  MoveL 175 to (-40.27, 47.68, 22.23) mm, rotated rx -180 ry 0 rz 180 deg; joints [-166.608, 53.388, -63.861, 166.389, 79.815, 2.452]
  Call Extruder(125.76334)
  MoveL 176 to (-40.23, 47.49, 22.22) mm, rotated rx 180 ry 0 rz -180 deg; joints [-166.656, 53.383, -63.865, 166.438, 79.804, 2.445]
  MoveL 177 to (-40.23, 47.49, 22.22) mm, rotated rx 180 ry 0 rz -180 deg; joints [-166.656, 53.383, -63.865, 166.438, 79.804, 2.445]
  Call Extruder(125.95387)
  MoveL 178 to (-40.2, 47.33, 22.22) mm, rotated rx -180 ry 0 rz -180 deg; joints [-166.699, 53.379, -63.869, 166.481, 79.794, 2.439]
  MoveL 179 to (-40.2, 47.33, 22.22) mm, rotated rx -180 ry 0 rz -180 deg; joints [-166.699, 53.379, -63.869, 166.481, 79.794, 2.439]
  Call Extruder(126.19017)
  MoveL 180 to (-40.15, 47.12, 22.22) mm, rotated rx -180 ry 0 rz 180 deg; joints [-166.751, 53.373, -63.874, 166.534, 79.782, 2.432]
  MoveL 181 to (-40.15, 47.12, 22.22) mm, rotated rx -180 ry 0 rz 180 deg; joints [-166.751, 53.373, -63.874, 166.534, 79.782, 2.432]
  Call Extruder(126.42754)
  MoveL 182 to (-40.11, 46.92, 22.22) mm, rotated rx -180 ry 0 rz -180 deg; joints [-166.804, 53.367, -63.878, 166.587, 79.77, 2.425]
  MoveL 183 to (-40.11, 46.92, 22.22) mm, rotated rx -180 ry 0 rz -180 deg; joints [-166.804, 53.367, -63.878, 166.587, 79.77, 2.425]
  Call Extruder(126.66598)
  MoveL 184 to (-40.06, 46.72, 22.23) mm, rotated rx 180 ry 0 rz -180 deg; joints [-166.857, 53.362, -63.883, 166.64, 79.758, 2.418]
  MoveL 185 to (-40.06, 46.72, 22.23) mm, rotated rx 180 ry 0 rz -180 deg; joints [-166.857, 53.362, -63.883, 166.64, 79.758, 2.418]
  Call Extruder(126.90549)
  MoveL 186 to (-40.02, 46.51, 22.22) mm, rotated rx -180 ry 0 rz 180 deg; joints [-166.909, 53.356, -63.887, 166.693, 79.745, 2.411]
  MoveL 187 to (-40.02, 46.51, 22.22) mm, rotated rx -180 ry 0 rz 180 deg; joints [-166.909, 53.356, -63.887, 166.693, 79.745, 2.411]
  Call Extruder(127.17442)
  MoveL 188 to (-39.95, 46.29, 22.22) mm, rotated rx -180 ry 0 rz -180 deg; joints [-166.966, 53.349, -63.893, 166.75, 79.73, 2.404]
  MoveL 189 to (-39.95, 46.29, 22.22) mm, rotated rx -180 ry 0 rz -180 deg; joints [-166.966, 53.349, -63.893, 166.75, 79.73, 2.404]
  Call Extruder(127.44468)
  MoveL 190 to (-39.88, 46.06, 22.22) mm, rotated rx 180 ry 0 rz 180 deg; joints [-167.022, 53.341, -63.899, 166.807, 79.715, 2.397]
  MoveL 191 to (-39.88, 46.06, 22.22) mm, rotated rx 180 ry 0 rz 180 deg; joints [-167.022, 53.341, -63.899, 166.807, 79.715, 2.397]
  Call Extruder(127.71628)
  MoveL 192 to (-39.82, 45.84, 22.22) mm, rotated rx 180 ry 0 rz -180 deg; joints [-167.079, 53.334, -63.905, 166.864, 79.7, 2.39]
  MoveL 193 to (-39.82, 45.84, 22.22) mm, rotated rx 180 ry 0 rz -180 deg; joints [-167.079, 53.334, -63.905, 166.864, 79.7, 2.39]
  Call Extruder(127.98921)
  MoveL 194 to (-39.75, 45.62, 22.22) mm, rotated rx 180 ry 0 rz -180 deg; joints [-167.136, 53.327, -63.911, 166.921, 79.684, 2.382]
  MoveL 195 to (-39.75, 45.62, 22.22) mm, rotated rx 180 ry 0 rz -180 deg; joints [-167.136, 53.327, -63.911, 166.921, 79.684, 2.382]
  Call Extruder(128.24265)
  MoveL 196 to (-39.68, 45.41, 22.22) mm, rotated rx -180 ry 0 rz 180 deg; joints [-167.188, 53.32, -63.916, 166.973, 79.67, 2.376]
  MoveL 197 to (-39.68, 45.41, 22.22) mm, rotated rx -180 ry 0 rz 180 deg; joints [-167.188, 53.32, -63.916, 166.973, 79.67, 2.376]
  Call Extruder(128.47637)
  MoveL 198 to (-39.62, 45.22, 22.22) mm, rotated rx 180 ry 0 rz 180 deg; joints [-167.235, 53.313, -63.922, 167.021, 79.657, 2.37]
  MoveL 199 to (-39.62, 45.22, 22.22) mm, rotated rx 180 ry 0 rz 180 deg; joints [-167.235, 53.313, -63.922, 167.021, 79.657, 2.37]
  Call Extruder(128.71114)
  MoveL 200 to (-39.56, 45.03, 22.22) mm, rotated rx 180 ry 0 rz 180 deg; joints [-167.283, 53.307, -63.927, 167.069, 79.644, 2.364]
  MoveL 201 to (-39.56, 45.03, 22.22) mm, rotated rx 180 ry 0 rz 180 deg; joints [-167.283, 53.307, -63.927, 167.069, 79.644, 2.364]
  Call Extruder(128.94697)
  MoveL 202 to (-39.5, 44.85, 22.22) mm, rotated rx -180 ry 0 rz 180 deg; joints [-167.331, 53.3, -63.932, 167.117, 79.63, 2.357]
  MoveL 203 to (-39.5, 44.85, 22.22) mm, rotated rx -180 ry 0 rz 180 deg; joints [-167.331, 53.3, -63.932, 167.117, 79.63, 2.357]
  Call Extruder(129.18384)
  MoveL 204 to (-39.44, 44.66, 22.22) mm, rotated rx -180 ry 0 rz 180 deg; joints [-167.379, 53.294, -63.937, 167.165, 79.617, 2.351]
  MoveL 205 to (-39.44, 44.66, 22.22) mm, rotated rx -180 ry 0 rz 180 deg; joints [-167.379, 53.294, -63.937, 167.165, 79.617, 2.351]
  Call Extruder(129.49225)
  MoveL 206 to (-39.35, 44.42, 22.23) mm, rotated rx -180 ry 0 rz 180 deg; joints [-167.439, 53.285, -63.944, 167.226, 79.599, 2.344]
  MoveL 207 to (-39.35, 44.42, 22.23) mm, rotated rx -180 ry 0 rz 180 deg; joints [-167.439, 53.285, -63.944, 167.226, 79.599, 2.344]
  Call Extruder(129.87335)
  MoveL 208 to (-39.22, 44.12, 22.22) mm, rotated rx 180 ry 0 rz 180 deg; joints [-167.512, 53.274, -63.953, 167.299, 79.576, 2.335]
  MoveL 209 to (-39.22, 44.12, 22.22) mm, rotated rx 180 ry 0 rz 180 deg; joints [-167.512, 53.274, -63.953, 167.299, 79.576, 2.335]
  Call Extruder(130.25623)
  MoveL 210 to (-39.11, 43.83, 22.22) mm, rotated rx -180 ry 0 rz -180 deg; joints [-167.584, 53.262, -63.962, 167.372, 79.553, 2.326]
  MoveL 211 to (-39.11, 43.83, 22.22) mm, rotated rx -180 ry 0 rz -180 deg; joints [-167.584, 53.262, -63.962, 167.372, 79.553, 2.326]
  Call Extruder(130.58614)
  MoveL 212 to (-39, 43.58, 22.22) mm, rotated rx 180 ry 0 rz -180 deg; joints [-167.646, 53.252, -63.97, 167.434, 79.533, 2.319]
  MoveL 213 to (-39, 43.58, 22.22) mm, rotated rx 180 ry 0 rz -180 deg; joints [-167.646, 53.252, -63.97, 167.434, 79.533, 2.319]
  Call Extruder(130.91747)
  MoveL 214 to (-38.89, 43.33, 22.22) mm, rotated rx -180 ry 0 rz 180 deg; joints [-167.708, 53.242, -63.978, 167.496, 79.513, 2.311]
  MoveL 215 to (-38.89, 43.33, 22.22) mm, rotated rx -180 ry 0 rz 180 deg; joints [-167.708, 53.242, -63.978, 167.496, 79.513, 2.311]
  Call Extruder(131.29867)
  MoveL 216 to (-38.75, 43.06, 22.22) mm, rotated rx -180 ry 0 rz 180 deg; joints [-167.776, 53.229, -63.988, 167.564, 79.488, 2.304]
  MoveL 217 to (-38.75, 43.06, 22.22) mm, rotated rx -180 ry 0 rz 180 deg; joints [-167.776, 53.229, -63.988, 167.564, 79.488, 2.304]
  Call Extruder(131.73146)
  MoveL 218 to (-38.57, 42.75, 22.22) mm, rotated rx -180 ry 0 rz -180 deg; joints [-167.849, 53.214, -64, 167.638, 79.459, 2.296]
  MoveL 219 to (-38.57, 42.75, 22.22) mm, rotated rx -180 ry 0 rz -180 deg; joints [-167.849, 53.214, -64, 167.638, 79.459, 2.296]
  Call Extruder(132.16610)
  MoveL 220 to (-38.4, 42.45, 22.22) mm, rotated rx -180 ry 0 rz -180 deg; joints [-167.923, 53.199, -64.011, 167.711, 79.43, 2.288]
  MoveL 221 to (-38.4, 42.45, 22.22) mm, rotated rx -180 ry 0 rz -180 deg; joints [-167.923, 53.199, -64.011, 167.711, 79.43, 2.288]
  Call Extruder(132.60257)
  MoveL 222 to (-38.22, 42.15, 22.22) mm, rotated rx -180 ry 0 rz 180 deg; joints [-167.997, 53.184, -64.023, 167.785, 79.401, 2.28]
  MoveL 223 to (-38.22, 42.15, 22.22) mm, rotated rx -180 ry 0 rz 180 deg; joints [-167.997, 53.184, -64.023, 167.785, 79.401, 2.28]
  Call Extruder(132.84952)
  MoveL 224 to (-38.12, 41.98, 22.22) mm, rotated rx 180 ry 0 rz 180 deg; joints [-168.038, 53.176, -64.03, 167.827, 79.385, 2.276]
  MoveL 225 to (-38.12, 41.98, 22.22) mm, rotated rx 180 ry 0 rz 180 deg; joints [-168.038, 53.176, -64.03, 167.827, 79.385, 2.276]
  Call Extruder(133.54809)
  MoveL 226 to (-37.79, 41.52, 22.23) mm, rotated rx 180 ry 0 rz -180 deg; joints [-168.144, 53.149, -64.05, 167.933, 79.334, 2.266]
  MoveL 227 to (-37.79, 41.52, 22.23) mm, rotated rx 180 ry 0 rz -180 deg; joints [-168.144, 53.149, -64.05, 167.933, 79.334, 2.266]
  Call Extruder(134.24946)
  MoveL 228 to (-37.47, 41.07, 22.22) mm, rotated rx -180 ry 0 rz 180 deg; joints [-168.25, 53.123, -64.07, 168.039, 79.284, 2.256]
  MoveL 229 to (-37.47, 41.07, 22.22) mm, rotated rx -180 ry 0 rz 180 deg; joints [-168.25, 53.123, -64.07, 168.039, 79.284, 2.256]
  Call Extruder(134.60151)
  MoveL 230 to (-37.3, 40.85, 22.22) mm, rotated rx -180 ry 0 rz -180 deg; joints [-168.304, 53.109, -64.081, 168.092, 79.259, 2.251]
  Call Extruder(136.34360)
  MoveL 231 to (-36.39, 39.81, 22.22) mm, rotated rx 180 ry 0 rz 180 deg; joints [-168.541, 53.038, -64.135, 168.329, 79.128, 2.231]
  Call Extruder(137.66925)
  MoveL 232 to (-35.61, 39.11, 22.22) mm, rotated rx -180 ry 0 rz -180 deg; joints [-168.693, 52.979, -64.179, 168.479, 79.021, 2.223]
  MoveL 233 to (-35.61, 39.11, 22.22) mm, rotated rx -180 ry 0 rz -180 deg; joints [-168.693, 52.979, -64.179, 168.479, 79.021, 2.223]
  Call Extruder(138.08410)
  MoveL 234 to (-35.35, 38.9, 22.22) mm, rotated rx 180 ry 0 rz 180 deg; joints [-168.739, 52.961, -64.193, 168.525, 78.987, 2.221]
  Call Extruder(138.78545)
  MoveL 235 to (-34.9, 38.57, 22.22) mm, rotated rx 180 ry 0 rz 180 deg; joints [-168.806, 52.928, -64.217, 168.591, 78.928, 2.219]
  MoveL 236 to (-34.9, 38.57, 22.22) mm, rotated rx 180 ry 0 rz 180 deg; joints [-168.806, 52.928, -64.217, 168.591, 78.928, 2.219]
  Call Extruder(139.48400)
  MoveL 237 to (-34.45, 38.24, 22.22) mm, rotated rx 180 ry 0 rz -180 deg; joints [-168.874, 52.895, -64.241, 168.658, 78.869, 2.217]
  MoveL 238 to (-34.45, 38.24, 22.22) mm, rotated rx 180 ry 0 rz -180 deg; joints [-168.874, 52.895, -64.241, 168.658, 78.869, 2.217]
  Call Extruder(139.86003)
  MoveL 239 to (-34.21, 38.07, 22.22) mm, rotated rx -180 ry 0 rz 180 deg; joints [-168.91, 52.877, -64.254, 168.694, 78.838, 2.217]
  MoveL 240 to (-34.21, 38.07, 22.22) mm, rotated rx -180 ry 0 rz 180 deg; joints [-168.91, 52.877, -64.254, 168.694, 78.838, 2.217]
  Call Extruder(140.29650)
  MoveL 241 to (-33.9, 37.89, 22.22) mm, rotated rx -180 ry 0 rz 180 deg; joints [-168.944, 52.855, -64.27, 168.726, 78.799, 2.217]
  MoveL 242 to (-33.9, 37.89, 22.22) mm, rotated rx -180 ry 0 rz 180 deg; joints [-168.944, 52.855, -64.27, 168.726, 78.799, 2.217]
  Call Extruder(140.73113)
  MoveL 243 to (-33.6, 37.71, 22.22) mm, rotated rx -180 ry 0 rz -180 deg; joints [-168.977, 52.833, -64.286, 168.758, 78.761, 2.218]
  MoveL 244 to (-33.6, 37.71, 22.22) mm, rotated rx -180 ry 0 rz -180 deg; joints [-168.977, 52.833, -64.286, 168.758, 78.761, 2.218]
  Call Extruder(141.16391)
  MoveL 245 to (-33.29, 37.54, 22.22) mm, rotated rx -180 ry 0 rz -180 deg; joints [-169.01, 52.812, -64.302, 168.791, 78.723, 2.219]
  MoveL 246 to (-33.29, 37.54, 22.22) mm, rotated rx -180 ry 0 rz -180 deg; joints [-169.01, 52.812, -64.302, 168.791, 78.723, 2.219]
  Call Extruder(141.59485)
  MoveL 247 to (-32.99, 37.36, 22.22) mm, rotated rx -180 ry 0 rz -180 deg; joints [-169.043, 52.79, -64.318, 168.823, 78.685, 2.22]
  MoveL 248 to (-32.99, 37.36, 22.22) mm, rotated rx -180 ry 0 rz -180 deg; joints [-169.043, 52.79, -64.318, 168.823, 78.685, 2.22]
  Call Extruder(141.92621)
  MoveL 249 to (-32.74, 37.26, 22.22) mm, rotated rx 180 ry 0 rz 180 deg; joints [-169.06, 52.772, -64.33, 168.839, 78.655, 2.223]
  MoveL 250 to (-32.74, 37.26, 22.22) mm, rotated rx 180 ry 0 rz 180 deg; joints [-169.06, 52.772, -64.33, 168.839, 78.655, 2.223]
  Call Extruder(142.25615)
  MoveL 251 to (-32.49, 37.15, 22.22) mm, rotated rx -180 ry 0 rz -180 deg; joints [-169.077, 52.755, -64.343, 168.855, 78.625, 2.225]
  MoveL 252 to (-32.49, 37.15, 22.22) mm, rotated rx -180 ry 0 rz -180 deg; joints [-169.077, 52.755, -64.343, 168.855, 78.625, 2.225]
  Call Extruder(142.61184)
  MoveL 253 to (-32.22, 37.03, 22.23) mm, rotated rx -180 ry 0 rz 180 deg; joints [-169.095, 52.736, -64.356, 168.872, 78.593, 2.228]
  MoveL 254 to (-32.22, 37.03, 22.23) mm, rotated rx -180 ry 0 rz 180 deg; joints [-169.095, 52.736, -64.356, 168.872, 78.593, 2.228]
  Call Extruder(142.99292)
  MoveL 255 to (-31.93, 36.91, 22.22) mm, rotated rx -180 ry 0 rz 180 deg; joints [-169.113, 52.716, -64.371, 168.89, 78.558, 2.231]
  MoveL 256 to (-31.93, 36.91, 22.22) mm, rotated rx -180 ry 0 rz 180 deg; joints [-169.113, 52.716, -64.371, 168.89, 78.558, 2.231]
  Call Extruder(143.37221)
  MoveL 257 to (-31.64, 36.79, 22.22) mm, rotated rx 180 ry 0 rz 180 deg; joints [-169.132, 52.695, -64.385, 168.907, 78.523, 2.234]
  MoveL 258 to (-31.64, 36.79, 22.22) mm, rotated rx 180 ry 0 rz 180 deg; joints [-169.132, 52.695, -64.385, 168.907, 78.523, 2.234]
  Call Extruder(143.60909)
  MoveL 259 to (-31.45, 36.73, 22.22) mm, rotated rx -180 ry 0 rz 180 deg; joints [-169.139, 52.682, -64.394, 168.914, 78.501, 2.237]
  MoveL 260 to (-31.45, 36.73, 22.22) mm, rotated rx -180 ry 0 rz 180 deg; joints [-169.139, 52.682, -64.394, 168.914, 78.501, 2.237]
  Call Extruder(143.84491)
  MoveL 261 to (-31.26, 36.67, 22.23) mm, rotated rx 180 ry 0 rz -180 deg; joints [-169.146, 52.669, -64.403, 168.92, 78.479, 2.24]
  MoveL 262 to (-31.26, 36.67, 22.23) mm, rotated rx 180 ry 0 rz -180 deg; joints [-169.146, 52.669, -64.403, 168.92, 78.479, 2.24]
  Call Extruder(144.07969)
  MoveL 263 to (-31.07, 36.61, 22.22) mm, rotated rx 180 ry 0 rz -180 deg; joints [-169.154, 52.656, -64.412, 168.927, 78.457, 2.243]
  MoveL 264 to (-31.07, 36.61, 22.22) mm, rotated rx 180 ry 0 rz -180 deg; joints [-169.154, 52.656, -64.412, 168.927, 78.457, 2.243]
  Call Extruder(144.31341)
  MoveL 265 to (-30.88, 36.55, 22.23) mm, rotated rx 180 ry 0 rz -180 deg; joints [-169.161, 52.643, -64.422, 168.933, 78.435, 2.246]
  MoveL 266 to (-30.88, 36.55, 22.23) mm, rotated rx 180 ry 0 rz -180 deg; joints [-169.161, 52.643, -64.422, 168.933, 78.435, 2.246]
  Call Extruder(144.54609)
  MoveL 267 to (-30.7, 36.49, 22.22) mm, rotated rx -180 ry 0 rz -180 deg; joints [-169.168, 52.63, -64.431, 168.94, 78.413, 2.248]
  MoveL 268 to (-30.7, 36.49, 22.22) mm, rotated rx -180 ry 0 rz -180 deg; joints [-169.168, 52.63, -64.431, 168.94, 78.413, 2.248]
  Call Extruder(144.81901)
  MoveL 269 to (-30.47, 36.42, 22.22) mm, rotated rx -180 ry 0 rz 180 deg; joints [-169.175, 52.615, -64.441, 168.946, 78.387, 2.252]
  MoveL 270 to (-30.47, 36.42, 22.22) mm, rotated rx -180 ry 0 rz 180 deg; joints [-169.175, 52.615, -64.441, 168.946, 78.387, 2.252]
  Call Extruder(145.09061)
  MoveL 271 to (-30.25, 36.35, 22.22) mm, rotated rx -180 ry 0 rz -180 deg; joints [-169.182, 52.599, -64.452, 168.952, 78.361, 2.256]
  MoveL 272 to (-30.25, 36.35, 22.22) mm, rotated rx -180 ry 0 rz -180 deg; joints [-169.182, 52.599, -64.452, 168.952, 78.361, 2.256]
  Call Extruder(145.36086)
  MoveL 273 to (-30.02, 36.28, 22.22) mm, rotated rx 180 ry 0 rz 180 deg; joints [-169.19, 52.584, -64.463, 168.959, 78.335, 2.259]
  MoveL 274 to (-30.02, 36.28, 22.22) mm, rotated rx 180 ry 0 rz 180 deg; joints [-169.19, 52.584, -64.463, 168.959, 78.335, 2.259]
  Call Extruder(145.62979)
  MoveL 275 to (-29.8, 36.22, 22.22) mm, rotated rx 180 ry 0 rz 180 deg; joints [-169.197, 52.568, -64.474, 168.965, 78.309, 2.263]
  MoveL 276 to (-29.8, 36.22, 22.22) mm, rotated rx 180 ry 0 rz 180 deg; joints [-169.197, 52.568, -64.474, 168.965, 78.309, 2.263]
  Call Extruder(145.88314)
  MoveL 277 to (-29.59, 36.16, 22.22) mm, rotated rx 180 ry 0 rz 180 deg; joints [-169.202, 52.553, -64.484, 168.969, 78.284, 2.267]
  MoveL 278 to (-29.59, 36.16, 22.22) mm, rotated rx 180 ry 0 rz 180 deg; joints [-169.202, 52.553, -64.484, 168.969, 78.284, 2.267]
  Call Extruder(146.12159)
  MoveL 279 to (-29.38, 36.12, 22.22) mm, rotated rx 180 ry 0 rz 180 deg; joints [-169.203, 52.54, -64.493, 168.97, 78.261, 2.271]
  MoveL 280 to (-29.38, 36.12, 22.22) mm, rotated rx 180 ry 0 rz 180 deg; joints [-169.203, 52.54, -64.493, 168.97, 78.261, 2.271]
  Call Extruder(146.35896)
  MoveL 281 to (-29.18, 36.07, 22.22) mm, rotated rx 180 ry 0 rz 180 deg; joints [-169.205, 52.526, -64.503, 168.97, 78.238, 2.275]
  MoveL 282 to (-29.18, 36.07, 22.22) mm, rotated rx 180 ry 0 rz 180 deg; joints [-169.205, 52.526, -64.503, 168.97, 78.238, 2.275]
  Call Extruder(146.59526)
  MoveL 283 to (-28.97, 36.03, 22.22) mm, rotated rx 180 ry 0 rz -180 deg; joints [-169.207, 52.512, -64.512, 168.971, 78.215, 2.28]
  MoveL 284 to (-28.97, 36.03, 22.22) mm, rotated rx 180 ry 0 rz -180 deg; joints [-169.207, 52.512, -64.512, 168.971, 78.215, 2.28]
  Call Extruder(146.83050)
  MoveL 285 to (-28.77, 35.98, 22.22) mm, rotated rx -180 ry 0 rz 180 deg; joints [-169.208, 52.498, -64.522, 168.972, 78.192, 2.284]
  MoveL 286 to (-28.77, 35.98, 22.22) mm, rotated rx -180 ry 0 rz 180 deg; joints [-169.208, 52.498, -64.522, 168.972, 78.192, 2.284]
  Call Extruder(147.11443)
  MoveL 287 to (-28.52, 35.93, 22.23) mm, rotated rx -180 ry 0 rz 180 deg; joints [-169.209, 52.481, -64.533, 168.972, 78.164, 2.289]
  MoveL 288 to (-28.52, 35.93, 22.23) mm, rotated rx -180 ry 0 rz 180 deg; joints [-169.209, 52.481, -64.533, 168.972, 78.164, 2.289]
  Call Extruder(147.39692)
  MoveL 289 to (-28.27, 35.88, 22.22) mm, rotated rx -180 ry 0 rz -180 deg; joints [-169.209, 52.464, -64.545, 168.971, 78.136, 2.295]
  MoveL 290 to (-28.27, 35.88, 22.22) mm, rotated rx -180 ry 0 rz -180 deg; joints [-169.209, 52.464, -64.545, 168.971, 78.136, 2.295]
  Call Extruder(147.67798)
  MoveL 291 to (-28.02, 35.83, 22.22) mm, rotated rx -180 ry 0 rz 180 deg; joints [-169.21, 52.447, -64.556, 168.97, 78.108, 2.3]
  MoveL 292 to (-28.02, 35.83, 22.22) mm, rotated rx -180 ry 0 rz 180 deg; joints [-169.21, 52.447, -64.556, 168.97, 78.108, 2.3]
  Call Extruder(147.95760)
  MoveL 293 to (-27.77, 35.78, 22.22) mm, rotated rx -180 ry 0 rz -180 deg; joints [-169.211, 52.43, -64.568, 168.97, 78.08, 2.306]
  MoveL 294 to (-27.77, 35.78, 22.22) mm, rotated rx -180 ry 0 rz -180 deg; joints [-169.211, 52.43, -64.568, 168.97, 78.08, 2.306]
  Call Extruder(148.23578)
  MoveL 295 to (-27.53, 35.73, 22.22) mm, rotated rx -180 ry 0 rz 180 deg; joints [-169.211, 52.413, -64.579, 168.969, 78.052, 2.311]
  MoveL 296 to (-27.53, 35.73, 22.22) mm, rotated rx -180 ry 0 rz 180 deg; joints [-169.211, 52.413, -64.579, 168.969, 78.052, 2.311]
  Call Extruder(148.51252)
  MoveL 297 to (-27.28, 35.68, 22.22) mm, rotated rx -180 ry 0 rz 180 deg; joints [-169.212, 52.395, -64.591, 168.969, 78.024, 2.317]
  MoveL 298 to (-27.28, 35.68, 22.22) mm, rotated rx -180 ry 0 rz 180 deg; joints [-169.212, 52.395, -64.591, 168.969, 78.024, 2.317]
  Call Extruder(148.72072)
  MoveL 299 to (-27.09, 35.65, 22.22) mm, rotated rx -180 ry 0 rz -180 deg; joints [-169.212, 52.383, -64.599, 168.968, 78.003, 2.321]
  MoveL 300 to (-27.09, 35.65, 22.22) mm, rotated rx -180 ry 0 rz -180 deg; joints [-169.212, 52.383, -64.599, 168.968, 78.003, 2.321]
  Call Extruder(148.95842)
  MoveL 301 to (-26.87, 35.61, 22.22) mm, rotated rx -180 ry 0 rz -180 deg; joints [-169.211, 52.368, -64.609, 168.966, 77.978, 2.326]
  MoveL 302 to (-26.87, 35.61, 22.22) mm, rotated rx -180 ry 0 rz -180 deg; joints [-169.211, 52.368, -64.609, 168.966, 77.978, 2.326]
  Call Extruder(149.29181)
  MoveL 303 to (-26.57, 35.56, 22.22) mm, rotated rx -180 ry 0 rz -180 deg; joints [-169.208, 52.347, -64.623, 168.962, 77.945, 2.333]
  MoveL 304 to (-26.57, 35.56, 22.22) mm, rotated rx -180 ry 0 rz -180 deg; joints [-169.208, 52.347, -64.623, 168.962, 77.945, 2.333]
  Call Extruder(149.62348)
  MoveL 305 to (-26.26, 35.51, 22.22) mm, rotated rx 180 ry 0 rz -180 deg; joints [-169.205, 52.326, -64.637, 168.957, 77.911, 2.341]
  MoveL 306 to (-26.26, 35.51, 22.22) mm, rotated rx 180 ry 0 rz -180 deg; joints [-169.205, 52.326, -64.637, 168.957, 77.911, 2.341]
  Call Extruder(149.95342)
  MoveL 307 to (-25.96, 35.47, 22.22) mm, rotated rx 180 ry 0 rz 180 deg; joints [-169.202, 52.305, -64.65, 168.953, 77.877, 2.348]
  MoveL 308 to (-25.96, 35.47, 22.22) mm, rotated rx 180 ry 0 rz 180 deg; joints [-169.202, 52.305, -64.65, 168.953, 77.877, 2.348]
  Call Extruder(150.28165)
  MoveL 309 to (-25.65, 35.42, 22.22) mm, rotated rx 180 ry 0 rz 180 deg; joints [-169.199, 52.284, -64.664, 168.948, 77.843, 2.355]
  MoveL 310 to (-25.65, 35.42, 22.22) mm, rotated rx 180 ry 0 rz 180 deg; joints [-169.199, 52.284, -64.664, 168.948, 77.843, 2.355]
  Call Extruder(150.60817)
  MoveL 311 to (-25.34, 35.37, 22.22) mm, rotated rx 180 ry 0 rz 180 deg; joints [-169.196, 52.263, -64.678, 168.944, 77.809, 2.363]
  MoveL 312 to (-25.34, 35.37, 22.22) mm, rotated rx 180 ry 0 rz 180 deg; joints [-169.196, 52.263, -64.678, 168.944, 77.809, 2.363]
  Call Extruder(150.97524)
  MoveL 313 to (-25, 35.32, 22.22) mm, rotated rx 180 ry 0 rz -180 deg; joints [-169.191, 52.239, -64.693, 168.937, 77.771, 2.372]
  MoveL 314 to (-25, 35.32, 22.22) mm, rotated rx 180 ry 0 rz -180 deg; joints [-169.191, 52.239, -64.693, 168.937, 77.771, 2.372]
  Call Extruder(151.38268)
  MoveL 315 to (-24.61, 35.27, 22.22) mm, rotated rx 180 ry 0 rz -180 deg; joints [-169.182, 52.213, -64.71, 168.926, 77.728, 2.382]
  MoveL 316 to (-24.61, 35.27, 22.22) mm, rotated rx 180 ry 0 rz -180 deg; joints [-169.182, 52.213, -64.71, 168.926, 77.728, 2.382]
  Call Extruder(151.78808)
  MoveL 317 to (-24.22, 35.23, 22.22) mm, rotated rx 180 ry 0 rz 180 deg; joints [-169.174, 52.186, -64.727, 168.916, 77.686, 2.392]
  MoveL 318 to (-24.22, 35.23, 22.22) mm, rotated rx 180 ry 0 rz 180 deg; joints [-169.174, 52.186, -64.727, 168.916, 77.686, 2.392]
  Call Extruder(152.19142)
  MoveL 319 to (-23.83, 35.18, 22.23) mm, rotated rx -180 ry 0 rz 180 deg; joints [-169.166, 52.16, -64.744, 168.905, 77.644, 2.403]
  MoveL 320 to (-23.83, 35.18, 22.23) mm, rotated rx -180 ry 0 rz 180 deg; joints [-169.166, 52.16, -64.744, 168.905, 77.644, 2.403]
  Call Extruder(152.59271)
  MoveL 321 to (-23.45, 35.14, 22.22) mm, rotated rx -180 ry 0 rz -180 deg; joints [-169.157, 52.133, -64.761, 168.895, 77.601, 2.413]
  MoveL 322 to (-23.45, 35.14, 22.22) mm, rotated rx -180 ry 0 rz -180 deg; joints [-169.157, 52.133, -64.761, 168.895, 77.601, 2.413]
  Call Extruder(153.19759)
  MoveL 323 to (-22.86, 35.09, 22.22) mm, rotated rx 180 ry 0 rz 180 deg; joints [-169.137, 52.093, -64.786, 168.871, 77.538, 2.431]
  MoveL 324 to (-22.86, 35.09, 22.22) mm, rotated rx 180 ry 0 rz 180 deg; joints [-169.137, 52.093, -64.786, 168.871, 77.538, 2.431]
  Call Extruder(153.79932)
  MoveL 325 to (-22.27, 35.05, 22.22) mm, rotated rx -180 ry 0 rz -180 deg; joints [-169.117, 52.053, -64.812, 168.848, 77.474, 2.448]
  MoveL 326 to (-22.27, 35.05, 22.22) mm, rotated rx -180 ry 0 rz -180 deg; joints [-169.117, 52.053, -64.812, 168.848, 77.474, 2.448]
  Call Extruder(154.39790)
  MoveL 327 to (-21.68, 35, 22.22) mm, rotated rx -180 ry 0 rz 180 deg; joints [-169.096, 52.012, -64.837, 168.824, 77.411, 2.466]
  MoveL 328 to (-21.68, 35, 22.22) mm, rotated rx -180 ry 0 rz 180 deg; joints [-169.096, 52.012, -64.837, 168.824, 77.411, 2.466]
  Call Extruder(155.56967)
  MoveL 329 to (-20.52, 34.95, 22.22) mm, rotated rx -180 ry 0 rz -180 deg; joints [-169.042, 51.933, -64.886, 168.763, 77.287, 2.503]
  MoveL 330 to (-20.52, 34.95, 22.22) mm, rotated rx -180 ry 0 rz -180 deg; joints [-169.042, 51.933, -64.886, 168.763, 77.287, 2.503]
  Call Extruder(157.02754)
  MoveL 331 to (-19.06, 34.91, 22.22) mm, rotated rx -180 ry 0 rz 180 deg; joints [-168.967, 51.833, -64.946, 168.68, 77.134, 2.552]
  Call Extruder(395.62063)
  MoveL 332 to (219.06, 34.91, 22.22) mm, rotated rx -180 ry 0 rz 180 deg; joints [-30.588, 42.292, -67.166, 33.086, 111.229, 13.274]
  Call Extruder(396.49572)
  MoveL 333 to (219.94, 34.93, 22.22) mm, rotated rx -180 ry 0 rz 180 deg; joints [-30.233, 42.366, -67.167, 32.701, 111.249, 13.098]
  MoveL 334 to (219.94, 34.93, 22.22) mm, rotated rx -180 ry 0 rz 180 deg; joints [-30.233, 42.366, -67.167, 32.701, 111.249, 13.098]
  Call Extruder(397.66749)
  MoveL 335 to (221.1, 34.98, 22.22) mm, rotated rx 180 ry 0 rz 180 deg; joints [-29.789, 42.465, -67.169, 32.215, 111.267, 12.874]
  MoveL 336 to (221.1, 34.98, 22.22) mm, rotated rx 180 ry 0 rz 180 deg; joints [-29.789, 42.465, -67.169, 32.215, 111.267, 12.874]
  Call Extruder(398.55557)
  MoveL 337 to (221.97, 35.02, 22.22) mm, rotated rx -180 ry 0 rz 180 deg; joints [-29.47, 42.541, -67.171, 31.867, 111.274, 12.711]
  MoveL 338 to (221.97, 35.02, 22.22) mm, rotated rx -180 ry 0 rz 180 deg; joints [-29.47, 42.541, -67.171, 31.867, 111.274, 12.711]
  Call Extruder(399.15730)
  MoveL 339 to (222.56, 35.07, 22.22) mm, rotated rx 180 ry 0 rz 180 deg; joints [-29.272, 42.592, -67.171, 31.649, 111.274, 12.606]
  MoveL 340 to (222.56, 35.07, 22.22) mm, rotated rx 180 ry 0 rz 180 deg; joints [-29.272, 42.592, -67.171, 31.649, 111.274, 12.606]
  Call Extruder(399.76217)
  MoveL 341 to (223.15, 35.11, 22.22) mm, rotated rx 180 ry 0 rz 180 deg; joints [-29.075, 42.644, -67.172, 31.432, 111.274, 12.503]
  MoveL 342 to (223.15, 35.11, 22.22) mm, rotated rx 180 ry 0 rz 180 deg; joints [-29.075, 42.644, -67.172, 31.432, 111.274, 12.503]
  Call Extruder(400.26672)
  MoveL 343 to (223.64, 35.16, 22.22) mm, rotated rx -180 ry 0 rz 180 deg; joints [-28.92, 42.687, -67.173, 31.261, 111.271, 12.42]
  MoveL 344 to (223.64, 35.16, 22.22) mm, rotated rx -180 ry 0 rz 180 deg; joints [-28.92, 42.687, -67.173, 31.261, 111.271, 12.42]
  Call Extruder(400.67007)
  MoveL 345 to (224.03, 35.21, 22.22) mm, rotated rx -180 ry 0 rz 180 deg; joints [-28.804, 42.722, -67.173, 31.133, 111.266, 12.357]
  MoveL 346 to (224.03, 35.21, 22.22) mm, rotated rx -180 ry 0 rz 180 deg; joints [-28.804, 42.722, -67.173, 31.133, 111.266, 12.357]
  Call Extruder(401.07546)
  MoveL 347 to (224.42, 35.25, 22.22) mm, rotated rx -180 ry 0 rz 180 deg; joints [-28.69, 42.757, -67.173, 31.006, 111.261, 12.294]
  MoveL 348 to (224.42, 35.25, 22.22) mm, rotated rx -180 ry 0 rz 180 deg; joints [-28.69, 42.757, -67.173, 31.006, 111.261, 12.294]
  Call Extruder(401.48291)
  MoveL 349 to (224.8, 35.3, 22.22) mm, rotated rx -180 ry 0 rz 180 deg; joints [-28.577, 42.792, -67.173, 30.88, 111.255, 12.232]
  MoveL 350 to (224.8, 35.3, 22.22) mm, rotated rx -180 ry 0 rz 180 deg; joints [-28.577, 42.792, -67.173, 30.88, 111.255, 12.232]
  Call Extruder(401.89240)
  MoveL 351 to (225.19, 35.34, 22.22) mm, rotated rx -180 ry 0 rz 180 deg; joints [-28.465, 42.826, -67.173, 30.756, 111.249, 12.171]
  MoveL 352 to (225.19, 35.34, 22.22) mm, rotated rx -180 ry 0 rz 180 deg; joints [-28.465, 42.826, -67.173, 30.756, 111.249, 12.171]
  Call Extruder(402.21894)
  MoveL 353 to (225.5, 35.39, 22.22) mm, rotated rx -180 ry 0 rz 180 deg; joints [-28.385, 42.854, -67.173, 30.667, 111.242, 12.125]
  MoveL 354 to (225.5, 35.39, 22.22) mm, rotated rx -180 ry 0 rz 180 deg; joints [-28.385, 42.854, -67.173, 30.667, 111.242, 12.125]
  Call Extruder(402.54719)
  MoveL 355 to (225.8, 35.44, 22.23) mm, rotated rx -180 ry 0 rz 180 deg; joints [-28.307, 42.882, -67.174, 30.579, 111.235, 12.08]
  MoveL 356 to (225.8, 35.44, 22.23) mm, rotated rx -180 ry 0 rz 180 deg; joints [-28.307, 42.882, -67.174, 30.579, 111.235, 12.08]
  Call Extruder(402.87716)
  MoveL 357 to (226.11, 35.49, 22.22) mm, rotated rx -180 ry 0 rz 180 deg; joints [-28.228, 42.91, -67.174, 30.492, 111.227, 12.035]
  MoveL 358 to (226.11, 35.49, 22.22) mm, rotated rx -180 ry 0 rz 180 deg; joints [-28.228, 42.91, -67.174, 30.492, 111.227, 12.035]
  Call Extruder(403.20885)
  MoveL 359 to (226.41, 35.54, 22.22) mm, rotated rx -180 ry 0 rz 180 deg; joints [-28.151, 42.938, -67.174, 30.405, 111.219, 11.991]
  MoveL 360 to (226.41, 35.54, 22.22) mm, rotated rx -180 ry 0 rz 180 deg; joints [-28.151, 42.938, -67.174, 30.405, 111.219, 11.991]
  Call Extruder(403.54226)
  MoveL 361 to (226.72, 35.59, 22.23) mm, rotated rx -180 ry 0 rz -180 deg; joints [-28.074, 42.966, -67.173, 30.318, 111.211, 11.946]
  MoveL 362 to (226.72, 35.59, 22.23) mm, rotated rx -180 ry 0 rz -180 deg; joints [-28.074, 42.966, -67.173, 30.318, 111.211, 11.946]
  Call Extruder(403.87738)
  MoveL 363 to (227.02, 35.63, 22.22) mm, rotated rx -180 ry 0 rz 180 deg; joints [-27.998, 42.994, -67.173, 30.234, 111.202, 11.902]
  MoveL 364 to (227.02, 35.63, 22.22) mm, rotated rx -180 ry 0 rz 180 deg; joints [-27.998, 42.994, -67.173, 30.234, 111.202, 11.902]
  Call Extruder(404.15384)
  MoveL 365 to (227.27, 35.68, 22.22) mm, rotated rx -180 ry 0 rz -180 deg; joints [-27.942, 43.017, -67.173, 30.171, 111.193, 11.869]
  MoveL 366 to (227.27, 35.68, 22.22) mm, rotated rx -180 ry 0 rz -180 deg; joints [-27.942, 43.017, -67.173, 30.171, 111.193, 11.869]
  Call Extruder(404.43174)
  MoveL 367 to (227.52, 35.73, 22.22) mm, rotated rx 180 ry 0 rz 180 deg; joints [-27.888, 43.04, -67.173, 30.109, 111.185, 11.835]
  MoveL 368 to (227.52, 35.73, 22.22) mm, rotated rx 180 ry 0 rz 180 deg; joints [-27.888, 43.04, -67.173, 30.109, 111.185, 11.835]
  Call Extruder(404.71108)
  MoveL 369 to (227.77, 35.78, 22.22) mm, rotated rx -180 ry 0 rz 180 deg; joints [-27.834, 43.063, -67.173, 30.048, 111.175, 11.802]
  MoveL 370 to (227.77, 35.78, 22.22) mm, rotated rx -180 ry 0 rz 180 deg; joints [-27.834, 43.063, -67.173, 30.048, 111.175, 11.802]
  Call Extruder(404.99186)
  MoveL 371 to (228.02, 35.83, 22.22) mm, rotated rx -180 ry 0 rz 180 deg; joints [-27.78, 43.087, -67.173, 29.986, 111.166, 11.769]
  MoveL 372 to (228.02, 35.83, 22.22) mm, rotated rx -180 ry 0 rz 180 deg; joints [-27.78, 43.087, -67.173, 29.986, 111.166, 11.769]
  Call Extruder(405.27408)
  MoveL 373 to (228.27, 35.88, 22.23) mm, rotated rx -180 ry 0 rz 180 deg; joints [-27.726, 43.11, -67.173, 29.926, 111.157, 11.736]
  MoveL 374 to (228.27, 35.88, 22.23) mm, rotated rx -180 ry 0 rz 180 deg; joints [-27.726, 43.11, -67.173, 29.926, 111.157, 11.736]
  Call Extruder(405.55775)
  MoveL 375 to (228.52, 35.93, 22.22) mm, rotated rx -180 ry 0 rz 180 deg; joints [-27.673, 43.133, -67.172, 29.865, 111.148, 11.704]
  MoveL 376 to (228.52, 35.93, 22.22) mm, rotated rx -180 ry 0 rz 180 deg; joints [-27.673, 43.133, -67.172, 29.865, 111.148, 11.704]
  Call Extruder(405.84286)
  MoveL 377 to (228.77, 35.98, 22.22) mm, rotated rx -180 ry 0 rz 180 deg; joints [-27.62, 43.156, -67.172, 29.805, 111.138, 11.671]
  MoveL 378 to (228.77, 35.98, 22.22) mm, rotated rx -180 ry 0 rz 180 deg; joints [-27.62, 43.156, -67.172, 29.805, 111.138, 11.671]
  Call Extruder(406.07863)
  MoveL 379 to (228.97, 36.03, 22.22) mm, rotated rx -180 ry 0 rz 180 deg; joints [-27.579, 43.175, -67.172, 29.758, 111.129, 11.645]
  MoveL 380 to (228.97, 36.03, 22.22) mm, rotated rx -180 ry 0 rz 180 deg; joints [-27.579, 43.175, -67.172, 29.758, 111.129, 11.645]
  Call Extruder(406.31548)
  MoveL 381 to (229.18, 36.07, 22.22) mm, rotated rx -180 ry 0 rz 180 deg; joints [-27.539, 43.194, -67.172, 29.712, 111.121, 11.62]
  MoveL 382 to (229.18, 36.07, 22.22) mm, rotated rx -180 ry 0 rz 180 deg; joints [-27.539, 43.194, -67.172, 29.712, 111.121, 11.62]
  Call Extruder(406.55339)
  MoveL 383 to (229.38, 36.12, 22.22) mm, rotated rx -180 ry 0 rz 180 deg; joints [-27.499, 43.213, -67.172, 29.666, 111.112, 11.594]
  MoveL 384 to (229.38, 36.12, 22.22) mm, rotated rx -180 ry 0 rz 180 deg; joints [-27.499, 43.213, -67.172, 29.666, 111.112, 11.594]
  Call Extruder(406.79238)
  MoveL 385 to (229.59, 36.16, 22.22) mm, rotated rx -180 ry 0 rz 180 deg; joints [-27.458, 43.233, -67.171, 29.62, 111.103, 11.569]
  MoveL 386 to (229.59, 36.16, 22.22) mm, rotated rx -180 ry 0 rz 180 deg; joints [-27.458, 43.233, -67.171, 29.62, 111.103, 11.569]
  Call Extruder(407.04637)
  MoveL 387 to (229.8, 36.22, 22.23) mm, rotated rx 180 ry 0 rz 180 deg; joints [-27.423, 43.253, -67.171, 29.579, 111.092, 11.544]
  MoveL 388 to (229.8, 36.22, 22.23) mm, rotated rx 180 ry 0 rz 180 deg; joints [-27.423, 43.253, -67.171, 29.579, 111.092, 11.544]
  Call Extruder(407.31597)
  MoveL 389 to (230.02, 36.28, 22.22) mm, rotated rx 180 ry 0 rz 180 deg; joints [-27.392, 43.275, -67.171, 29.542, 111.079, 11.521]
  MoveL 390 to (230.02, 36.28, 22.22) mm, rotated rx 180 ry 0 rz 180 deg; joints [-27.392, 43.275, -67.171, 29.542, 111.079, 11.521]
  Call Extruder(407.58690)
  MoveL 391 to (230.25, 36.35, 22.22) mm, rotated rx -180 ry 0 rz 180 deg; joints [-27.361, 43.297, -67.17, 29.506, 111.066, 11.498]
  MoveL 392 to (230.25, 36.35, 22.22) mm, rotated rx -180 ry 0 rz 180 deg; joints [-27.361, 43.297, -67.17, 29.506, 111.066, 11.498]
  Call Extruder(407.85917)
  MoveL 393 to (230.47, 36.42, 22.22) mm, rotated rx -180 ry 0 rz 180 deg; joints [-27.33, 43.318, -67.17, 29.469, 111.053, 11.474]
  MoveL 394 to (230.47, 36.42, 22.22) mm, rotated rx -180 ry 0 rz 180 deg; joints [-27.33, 43.318, -67.17, 29.469, 111.053, 11.474]
  Call Extruder(408.13278)
  MoveL 395 to (230.7, 36.49, 22.23) mm, rotated rx -180 ry 0 rz 180 deg; joints [-27.299, 43.34, -67.17, 29.432, 111.04, 11.451]
  MoveL 396 to (230.7, 36.49, 22.23) mm, rotated rx -180 ry 0 rz 180 deg; joints [-27.299, 43.34, -67.17, 29.432, 111.04, 11.451]
  Call Extruder(408.36597)
  MoveL 397 to (230.88, 36.55, 22.22) mm, rotated rx 180 ry 0 rz 180 deg; joints [-27.276, 43.359, -67.169, 29.405, 111.028, 11.433]
  MoveL 398 to (230.88, 36.55, 22.22) mm, rotated rx 180 ry 0 rz 180 deg; joints [-27.276, 43.359, -67.169, 29.405, 111.028, 11.433]
  Call Extruder(408.60021)
  MoveL 399 to (231.07, 36.61, 22.23) mm, rotated rx 180 ry 0 rz 180 deg; joints [-27.253, 43.377, -67.169, 29.377, 111.016, 11.414]
  MoveL 400 to (231.07, 36.61, 22.23) mm, rotated rx 180 ry 0 rz 180 deg; joints [-27.253, 43.377, -67.169, 29.377, 111.016, 11.414]
  Call Extruder(408.83551)
  MoveL 401 to (231.26, 36.67, 22.22) mm, rotated rx 180 ry 0 rz 180 deg; joints [-27.231, 43.396, -67.168, 29.35, 111.004, 11.396]
  MoveL 402 to (231.26, 36.67, 22.22) mm, rotated rx 180 ry 0 rz 180 deg; joints [-27.231, 43.396, -67.168, 29.35, 111.004, 11.396]
  Call Extruder(409.07185)
  MoveL 403 to (231.45, 36.73, 22.22) mm, rotated rx -180 ry 0 rz -180 deg; joints [-27.208, 43.414, -67.168, 29.322, 110.992, 11.377]
  MoveL 404 to (231.45, 36.73, 22.22) mm, rotated rx -180 ry 0 rz -180 deg; joints [-27.208, 43.414, -67.168, 29.322, 110.992, 11.377]
  Call Extruder(409.30925)
  MoveL 405 to (231.64, 36.79, 22.23) mm, rotated rx -180 ry 0 rz 180 deg; joints [-27.185, 43.432, -67.168, 29.295, 110.98, 11.359]
  MoveL 406 to (231.64, 36.79, 22.23) mm, rotated rx -180 ry 0 rz 180 deg; joints [-27.185, 43.432, -67.168, 29.295, 110.98, 11.359]
  Call Extruder(409.68944)
  MoveL 407 to (231.93, 36.91, 22.22) mm, rotated rx 180 ry 0 rz 180 deg; joints [-27.167, 43.462, -67.167, 29.27, 110.957, 11.336]
  MoveL 408 to (231.93, 36.91, 22.22) mm, rotated rx 180 ry 0 rz 180 deg; joints [-27.167, 43.462, -67.167, 29.27, 110.957, 11.336]
  Call Extruder(410.07143)
  MoveL 409 to (232.22, 37.04, 22.22) mm, rotated rx -180 ry 0 rz 180 deg; joints [-27.149, 43.492, -67.166, 29.245, 110.934, 11.313]
  MoveL 410 to (232.22, 37.04, 22.22) mm, rotated rx -180 ry 0 rz 180 deg; joints [-27.149, 43.492, -67.166, 29.245, 110.934, 11.313]
  Call Extruder(410.42789)
  MoveL 411 to (232.49, 37.15, 22.23) mm, rotated rx -180 ry 0 rz 180 deg; joints [-27.133, 43.519, -67.166, 29.224, 110.913, 11.293]
  MoveL 412 to (232.49, 37.15, 22.23) mm, rotated rx -180 ry 0 rz 180 deg; joints [-27.133, 43.519, -67.166, 29.224, 110.913, 11.293]
  Call Extruder(410.75854)
  MoveL 413 to (232.74, 37.26, 22.22) mm, rotated rx -180 ry 0 rz 180 deg; joints [-27.121, 43.545, -67.165, 29.206, 110.892, 11.274]
  MoveL 414 to (232.74, 37.26, 22.22) mm, rotated rx -180 ry 0 rz 180 deg; joints [-27.121, 43.545, -67.165, 29.206, 110.892, 11.274]
  Call Extruder(411.09062)
  MoveL 415 to (232.99, 37.36, 22.22) mm, rotated rx 180 ry 0 rz 180 deg; joints [-27.108, 43.57, -67.164, 29.187, 110.872, 11.256]
  MoveL 416 to (232.99, 37.36, 22.22) mm, rotated rx 180 ry 0 rz 180 deg; joints [-27.108, 43.57, -67.164, 29.187, 110.872, 11.256]
  Call Extruder(411.52249)
  MoveL 417 to (233.29, 37.54, 22.22) mm, rotated rx -180 ry 0 rz 180 deg; joints [-27.12, 43.603, -67.163, 29.193, 110.84, 11.242]
  MoveL 418 to (233.29, 37.54, 22.22) mm, rotated rx -180 ry 0 rz 180 deg; joints [-27.12, 43.603, -67.163, 29.193, 110.84, 11.242]
  Call Extruder(411.95620)
  MoveL 419 to (233.6, 37.71, 22.22) mm, rotated rx 180 ry 0 rz 180 deg; joints [-27.132, 43.636, -67.162, 29.2, 110.808, 11.229]
  MoveL 420 to (233.6, 37.71, 22.22) mm, rotated rx 180 ry 0 rz 180 deg; joints [-27.132, 43.636, -67.162, 29.2, 110.808, 11.229]
  Call Extruder(412.39175)
  MoveL 421 to (233.9, 37.89, 22.22) mm, rotated rx -180 ry 0 rz 180 deg; joints [-27.144, 43.669, -67.161, 29.206, 110.776, 11.216]
  MoveL 422 to (233.9, 37.89, 22.22) mm, rotated rx -180 ry 0 rz 180 deg; joints [-27.144, 43.669, -67.161, 29.206, 110.776, 11.216]
  Call Extruder(412.82915)
  MoveL 423 to (234.21, 38.06, 22.22) mm, rotated rx -180 ry 0 rz 180 deg; joints [-27.156, 43.702, -67.16, 29.213, 110.744, 11.203]
  MoveL 424 to (234.21, 38.06, 22.22) mm, rotated rx -180 ry 0 rz 180 deg; joints [-27.156, 43.702, -67.16, 29.213, 110.744, 11.203]
  Call Extruder(413.20589)
  MoveL 425 to (234.45, 38.24, 22.22) mm, rotated rx 180 ry 0 rz -180 deg; joints [-27.187, 43.73, -67.159, 29.24, 110.713, 11.199]
  MoveL 426 to (234.45, 38.24, 22.22) mm, rotated rx 180 ry 0 rz -180 deg; joints [-27.187, 43.73, -67.159, 29.24, 110.713, 11.199]
  Call Extruder(413.90582)
  MoveL 427 to (234.9, 38.57, 22.22) mm, rotated rx -180 ry 0 rz 180 deg; joints [-27.245, 43.782, -67.157, 29.291, 110.655, 11.193]
  MoveL 428 to (234.9, 38.57, 22.22) mm, rotated rx -180 ry 0 rz 180 deg; joints [-27.245, 43.782, -67.157, 29.291, 110.655, 11.193]
  Call Extruder(414.60855)
  MoveL 429 to (235.35, 38.9, 22.22) mm, rotated rx -180 ry 0 rz 180 deg; joints [-27.302, 43.833, -67.155, 29.341, 110.597, 11.186]
  Call Extruder(416.34741)
  MoveL 430 to (236.39, 39.81, 22.22) mm, rotated rx 180 ry 0 rz 180 deg; joints [-27.525, 43.958, -67.15, 29.55, 110.44, 11.199]
  Call Extruder(418.08626)
  MoveL 431 to (237.3, 40.85, 22.22) mm, rotated rx -180 ry 0 rz -180 deg; joints [-27.851, 44.078, -67.144, 29.869, 110.267, 11.251]
  Call Extruder(418.43762)
  MoveL 432 to (237.47, 41.07, 22.22) mm, rotated rx -180 ry 0 rz 180 deg; joints [-27.932, 44.102, -67.143, 29.948, 110.23, 11.268]
  MoveL 433 to (237.47, 41.07, 22.22) mm, rotated rx -180 ry 0 rz 180 deg; joints [-27.932, 44.102, -67.143, 29.948, 110.23, 11.268]
  Call Extruder(419.13755)
  MoveL 434 to (237.79, 41.52, 22.22) mm, rotated rx 180 ry 0 rz 180 deg; joints [-28.091, 44.148, -67.14, 30.106, 110.157, 11.299]
  MoveL 435 to (237.79, 41.52, 22.22) mm, rotated rx 180 ry 0 rz 180 deg; joints [-28.091, 44.148, -67.14, 30.106, 110.157, 11.299]
  Call Extruder(419.83467)
  MoveL 436 to (238.12, 41.97, 22.22) mm, rotated rx -180 ry 0 rz 180 deg; joints [-28.249, 44.195, -67.138, 30.261, 110.083, 11.329]
  MoveL 437 to (238.12, 41.97, 22.22) mm, rotated rx -180 ry 0 rz 180 deg; joints [-28.249, 44.195, -67.138, 30.261, 110.083, 11.329]
  Call Extruder(420.08158)
  MoveL 438 to (238.22, 42.15, 22.22) mm, rotated rx -180 ry 0 rz -180 deg; joints [-28.315, 44.21, -67.137, 30.328, 110.056, 11.344]
  MoveL 439 to (238.22, 42.15, 22.22) mm, rotated rx -180 ry 0 rz -180 deg; joints [-28.315, 44.21, -67.137, 30.328, 110.056, 11.344]
  Call Extruder(420.51713)
  MoveL 440 to (238.4, 42.45, 22.22) mm, rotated rx -180 ry 0 rz -180 deg; joints [-28.434, 44.238, -67.135, 30.446, 110.007, 11.371]
  MoveL 441 to (238.4, 42.45, 22.22) mm, rotated rx -180 ry 0 rz -180 deg; joints [-28.434, 44.238, -67.135, 30.446, 110.007, 11.371]
  Call Extruder(420.95084)
  MoveL 442 to (238.57, 42.75, 22.22) mm, rotated rx -180 ry 0 rz 180 deg; joints [-28.552, 44.266, -67.133, 30.563, 109.959, 11.397]
  MoveL 443 to (238.57, 42.75, 22.22) mm, rotated rx -180 ry 0 rz 180 deg; joints [-28.552, 44.266, -67.133, 30.563, 109.959, 11.397]
  Call Extruder(421.38271)
  MoveL 444 to (238.75, 43.06, 22.22) mm, rotated rx 180 ry 0 rz -180 deg; joints [-28.669, 44.293, -67.132, 30.68, 109.911, 11.423]
  MoveL 445 to (238.75, 43.06, 22.22) mm, rotated rx 180 ry 0 rz -180 deg; joints [-28.669, 44.293, -67.132, 30.68, 109.911, 11.423]
  Call Extruder(421.76312)
  MoveL 446 to (238.89, 43.33, 22.23) mm, rotated rx -180 ry 0 rz 180 deg; joints [-28.78, 44.317, -67.13, 30.792, 109.867, 11.448]
  MoveL 447 to (238.89, 43.33, 22.23) mm, rotated rx -180 ry 0 rz 180 deg; joints [-28.78, 44.317, -67.13, 30.792, 109.867, 11.448]
  Call Extruder(422.09380)
  MoveL 448 to (239, 43.58, 22.22) mm, rotated rx 180 ry 0 rz 180 deg; joints [-28.886, 44.337, -67.129, 30.898, 109.828, 11.474]
  MoveL 449 to (239, 43.58, 22.22) mm, rotated rx 180 ry 0 rz 180 deg; joints [-28.886, 44.337, -67.129, 30.898, 109.828, 11.474]
  Call Extruder(422.42305)
  MoveL 450 to (239.1, 43.83, 22.22) mm, rotated rx 180 ry 0 rz 180 deg; joints [-28.991, 44.356, -67.128, 31.004, 109.789, 11.5]
  MoveL 451 to (239.1, 43.83, 22.22) mm, rotated rx 180 ry 0 rz 180 deg; joints [-28.991, 44.356, -67.128, 31.004, 109.789, 11.5]
  Call Extruder(422.80503)
  MoveL 452 to (239.22, 44.12, 22.22) mm, rotated rx -180 ry 0 rz 180 deg; joints [-29.116, 44.379, -67.126, 31.129, 109.743, 11.531]
  MoveL 453 to (239.22, 44.12, 22.22) mm, rotated rx -180 ry 0 rz 180 deg; joints [-29.116, 44.379, -67.126, 31.129, 109.743, 11.531]
  Call Extruder(423.18522)
  MoveL 454 to (239.35, 44.42, 22.22) mm, rotated rx -180 ry 0 rz 180 deg; joints [-29.24, 44.402, -67.125, 31.253, 109.697, 11.561]
  MoveL 455 to (239.35, 44.42, 22.22) mm, rotated rx -180 ry 0 rz 180 deg; joints [-29.24, 44.402, -67.125, 31.253, 109.697, 11.561]
  Call Extruder(423.49290)
  MoveL 456 to (239.44, 44.66, 22.23) mm, rotated rx -180 ry 0 rz 180 deg; joints [-29.343, 44.42, -67.124, 31.358, 109.66, 11.586]
  MoveL 457 to (239.44, 44.66, 22.23) mm, rotated rx -180 ry 0 rz 180 deg; joints [-29.343, 44.42, -67.124, 31.358, 109.66, 11.586]
  Call Extruder(423.72925)
  MoveL 458 to (239.5, 44.85, 22.22) mm, rotated rx -180 ry 0 rz 180 deg; joints [-29.428, 44.434, -67.123, 31.443, 109.631, 11.608]
  MoveL 459 to (239.5, 44.85, 22.22) mm, rotated rx -180 ry 0 rz 180 deg; joints [-29.428, 44.434, -67.123, 31.443, 109.631, 11.608]
  Call Extruder(423.96455)
  MoveL 460 to (239.56, 45.03, 22.22) mm, rotated rx -180 ry 0 rz 180 deg; joints [-29.512, 44.447, -67.122, 31.527, 109.602, 11.629]
  MoveL 461 to (239.56, 45.03, 22.22) mm, rotated rx -180 ry 0 rz 180 deg; joints [-29.512, 44.447, -67.122, 31.527, 109.602, 11.629]
  Call Extruder(424.19880)
  MoveL 462 to (239.62, 45.22, 22.22) mm, rotated rx -180 ry 0 rz 180 deg; joints [-29.596, 44.461, -67.121, 31.612, 109.573, 11.651]
  MoveL 463 to (239.62, 45.22, 22.22) mm, rotated rx -180 ry 0 rz 180 deg; joints [-29.596, 44.461, -67.121, 31.612, 109.573, 11.651]
  Call Extruder(424.43200)
  MoveL 464 to (239.68, 45.41, 22.22) mm, rotated rx -180 ry 0 rz -180 deg; joints [-29.679, 44.474, -67.12, 31.696, 109.544, 11.672]
  MoveL 465 to (239.68, 45.41, 22.22) mm, rotated rx -180 ry 0 rz -180 deg; joints [-29.679, 44.474, -67.12, 31.696, 109.544, 11.672]
  Call Extruder(424.68486)
  MoveL 466 to (239.75, 45.62, 22.22) mm, rotated rx -180 ry 0 rz -180 deg; joints [-29.77, 44.489, -67.119, 31.788, 109.512, 11.695]
  MoveL 467 to (239.75, 45.62, 22.22) mm, rotated rx -180 ry 0 rz -180 deg; joints [-29.77, 44.489, -67.119, 31.788, 109.512, 11.695]
  Call Extruder(424.95712)
  MoveL 468 to (239.82, 45.84, 22.22) mm, rotated rx 180 ry 0 rz 180 deg; joints [-29.871, 44.504, -67.118, 31.889, 109.477, 11.72]
  MoveL 469 to (239.82, 45.84, 22.22) mm, rotated rx 180 ry 0 rz 180 deg; joints [-29.871, 44.504, -67.118, 31.889, 109.477, 11.72]
  Call Extruder(425.22805)
  MoveL 470 to (239.88, 46.06, 22.22) mm, rotated rx -180 ry 0 rz 180 deg; joints [-29.97, 44.52, -67.117, 31.989, 109.443, 11.745]
  MoveL 471 to (239.88, 46.06, 22.22) mm, rotated rx -180 ry 0 rz 180 deg; joints [-29.97, 44.52, -67.117, 31.989, 109.443, 11.745]
  Call Extruder(425.49763)
  MoveL 472 to (239.95, 46.29, 22.22) mm, rotated rx -180 ry 0 rz 180 deg; joints [-30.069, 44.535, -67.115, 32.089, 109.408, 11.77]
  MoveL 473 to (239.95, 46.29, 22.22) mm, rotated rx -180 ry 0 rz 180 deg; joints [-30.069, 44.535, -67.115, 32.089, 109.408, 11.77]
  Call Extruder(425.76589)
  MoveL 474 to (240.02, 46.51, 22.22) mm, rotated rx -180 ry 0 rz 180 deg; joints [-30.168, 44.551, -67.114, 32.189, 109.374, 11.794]
  MoveL 475 to (240.02, 46.51, 22.22) mm, rotated rx -180 ry 0 rz 180 deg; joints [-30.168, 44.551, -67.114, 32.189, 109.374, 11.794]
  Call Extruder(426.00483)
  MoveL 476 to (240.06, 46.72, 22.22) mm, rotated rx -180 ry 0 rz 180 deg; joints [-30.263, 44.564, -67.113, 32.285, 109.343, 11.819]
  MoveL 477 to (240.06, 46.72, 22.22) mm, rotated rx -180 ry 0 rz 180 deg; joints [-30.263, 44.564, -67.113, 32.285, 109.343, 11.819]
  Call Extruder(426.24270)
  MoveL 478 to (240.11, 46.92, 22.22) mm, rotated rx -180 ry 0 rz 180 deg; joints [-30.358, 44.577, -67.112, 32.38, 109.311, 11.844]
  MoveL 479 to (240.11, 46.92, 22.22) mm, rotated rx -180 ry 0 rz 180 deg; joints [-30.358, 44.577, -67.112, 32.38, 109.311, 11.844]
  Call Extruder(426.47950)
  MoveL 480 to (240.15, 47.12, 22.22) mm, rotated rx -180 ry 0 rz -180 deg; joints [-30.453, 44.59, -67.111, 32.476, 109.28, 11.868]
  MoveL 481 to (240.15, 47.12, 22.22) mm, rotated rx -180 ry 0 rz -180 deg; joints [-30.453, 44.59, -67.111, 32.476, 109.28, 11.868]
  Call Extruder(426.71523)
  MoveL 482 to (240.2, 47.33, 22.22) mm, rotated rx 180 ry 0 rz -180 deg; joints [-30.548, 44.603, -67.11, 32.571, 109.249, 11.893]
  MoveL 483 to (240.2, 47.33, 22.22) mm, rotated rx 180 ry 0 rz -180 deg; joints [-30.548, 44.603, -67.11, 32.571, 109.249, 11.893]
  Call Extruder(426.97511)
  MoveL 484 to (240.24, 47.56, 22.22) mm, rotated rx 180 ry 0 rz -180 deg; joints [-30.653, 44.617, -67.109, 32.677, 109.214, 11.92]
  MoveL 485 to (240.24, 47.56, 22.22) mm, rotated rx 180 ry 0 rz -180 deg; joints [-30.653, 44.617, -67.109, 32.677, 109.214, 11.92]
  Call Extruder(427.25877)
  MoveL 486 to (240.29, 47.8, 22.22) mm, rotated rx 180 ry 0 rz 180 deg; joints [-30.768, 44.633, -67.108, 32.794, 109.176, 11.95]
  MoveL 487 to (240.29, 47.8, 22.22) mm, rotated rx 180 ry 0 rz 180 deg; joints [-30.768, 44.633, -67.108, 32.794, 109.176, 11.95]
  Call Extruder(427.54099)
  MoveL 488 to (240.34, 48.05, 22.22) mm, rotated rx -180 ry 0 rz 180 deg; joints [-30.884, 44.648, -67.107, 32.911, 109.138, 11.979]
  MoveL 489 to (240.34, 48.05, 22.22) mm, rotated rx -180 ry 0 rz 180 deg; joints [-30.884, 44.648, -67.107, 32.911, 109.138, 11.979]
  Call Extruder(427.82177)
  MoveL 490 to (240.39, 48.3, 22.22) mm, rotated rx -180 ry 0 rz 180 deg; joints [-30.999, 44.664, -67.106, 33.027, 109.1, 12.009]
  MoveL 491 to (240.39, 48.3, 22.22) mm, rotated rx -180 ry 0 rz 180 deg; joints [-30.999, 44.664, -67.106, 33.027, 109.1, 12.009]
  Call Extruder(428.10111)
  MoveL 492 to (240.44, 48.55, 22.22) mm, rotated rx -180 ry 0 rz 180 deg; joints [-31.114, 44.68, -67.104, 33.142, 109.062, 12.038]
  MoveL 493 to (240.44, 48.55, 22.22) mm, rotated rx -180 ry 0 rz 180 deg; joints [-31.114, 44.68, -67.104, 33.142, 109.062, 12.038]
  Call Extruder(428.37901)
  MoveL 494 to (240.49, 48.8, 22.22) mm, rotated rx 180 ry 0 rz 180 deg; joints [-31.228, 44.695, -67.103, 33.257, 109.024, 12.067]
  MoveL 495 to (240.49, 48.8, 22.22) mm, rotated rx 180 ry 0 rz 180 deg; joints [-31.228, 44.695, -67.103, 33.257, 109.024, 12.067]
  Call Extruder(428.65546)
  MoveL 496 to (240.54, 49.05, 22.22) mm, rotated rx -180 ry 0 rz 180 deg; joints [-31.342, 44.711, -67.102, 33.372, 108.986, 12.095]
  MoveL 497 to (240.54, 49.05, 22.22) mm, rotated rx -180 ry 0 rz 180 deg; joints [-31.342, 44.711, -67.102, 33.372, 108.986, 12.095]
  Call Extruder(428.96049)
  MoveL 498 to (240.59, 49.33, 22.22) mm, rotated rx 180 ry 0 rz 180 deg; joints [-31.47, 44.728, -67.101, 33.501, 108.944, 12.127]
  MoveL 499 to (240.59, 49.33, 22.22) mm, rotated rx 180 ry 0 rz 180 deg; joints [-31.47, 44.728, -67.101, 33.501, 108.944, 12.127]
  Call Extruder(429.29393)
  MoveL 500 to (240.64, 49.63, 22.22) mm, rotated rx 180 ry 0 rz -180 deg; joints [-31.612, 44.746, -67.099, 33.644, 108.897, 12.163]
  MoveL 501 to (240.64, 49.63, 22.22) mm, rotated rx 180 ry 0 rz -180 deg; joints [-31.612, 44.746, -67.099, 33.644, 108.897, 12.163]
  Call Extruder(429.62565)
  MoveL 502 to (240.69, 49.94, 22.23) mm, rotated rx -180 ry 0 rz 180 deg; joints [-31.755, 44.765, -67.097, 33.787, 108.851, 12.199]
  MoveL 503 to (240.69, 49.94, 22.23) mm, rotated rx -180 ry 0 rz 180 deg; joints [-31.755, 44.765, -67.097, 33.787, 108.851, 12.199]
  Call Extruder(429.95564)
  MoveL 504 to (240.73, 50.24, 22.22) mm, rotated rx -180 ry 0 rz 180 deg; joints [-31.895, 44.783, -67.096, 33.929, 108.804, 12.234]
  MoveL 505 to (240.73, 50.24, 22.22) mm, rotated rx -180 ry 0 rz 180 deg; joints [-31.895, 44.783, -67.096, 33.929, 108.804, 12.234]
  Call Extruder(430.28392)
  MoveL 506 to (240.78, 50.55, 22.22) mm, rotated rx 180 ry 0 rz 180 deg; joints [-32.036, 44.802, -67.094, 34.07, 108.758, 12.269]
  MoveL 507 to (240.78, 50.55, 22.22) mm, rotated rx 180 ry 0 rz 180 deg; joints [-32.036, 44.802, -67.094, 34.07, 108.758, 12.269]
  Call Extruder(430.61048)
  MoveL 508 to (240.83, 50.86, 22.22) mm, rotated rx -180 ry 0 rz 180 deg; joints [-32.176, 44.82, -67.093, 34.211, 108.711, 12.304]
  MoveL 509 to (240.83, 50.86, 22.22) mm, rotated rx -180 ry 0 rz 180 deg; joints [-32.176, 44.82, -67.093, 34.211, 108.711, 12.304]
  Call Extruder(430.97758)
  MoveL 510 to (240.88, 51.2, 22.23) mm, rotated rx -180 ry 0 rz -180 deg; joints [-32.337, 44.841, -67.091, 34.372, 108.659, 12.344]
  MoveL 511 to (240.88, 51.2, 22.23) mm, rotated rx -180 ry 0 rz -180 deg; joints [-32.337, 44.841, -67.091, 34.372, 108.659, 12.344]
  Call Extruder(431.38502)
  MoveL 512 to (240.93, 51.59, 22.22) mm, rotated rx -180 ry 0 rz 180 deg; joints [-32.518, 44.863, -67.089, 34.554, 108.6, 12.389]
  MoveL 513 to (240.93, 51.59, 22.22) mm, rotated rx -180 ry 0 rz 180 deg; joints [-32.518, 44.863, -67.089, 34.554, 108.6, 12.389]
  Call Extruder(431.79041)
  MoveL 514 to (240.97, 51.98, 22.22) mm, rotated rx -180 ry 0 rz 180 deg; joints [-32.697, 44.886, -67.087, 34.734, 108.541, 12.433]
  MoveL 515 to (240.97, 51.98, 22.22) mm, rotated rx -180 ry 0 rz 180 deg; joints [-32.697, 44.886, -67.087, 34.734, 108.541, 12.433]
  Call Extruder(432.19375)
  MoveL 516 to (241.02, 52.36, 22.22) mm, rotated rx -180 ry 0 rz 180 deg; joints [-32.876, 44.908, -67.085, 34.914, 108.482, 12.477]
  MoveL 517 to (241.02, 52.36, 22.22) mm, rotated rx -180 ry 0 rz 180 deg; joints [-32.876, 44.908, -67.085, 34.914, 108.482, 12.477]
  Call Extruder(432.59504)
  MoveL 518 to (241.06, 52.75, 22.22) mm, rotated rx -180 ry 0 rz 180 deg; joints [-33.055, 44.931, -67.083, 35.093, 108.423, 12.52]
  MoveL 519 to (241.06, 52.75, 22.22) mm, rotated rx -180 ry 0 rz 180 deg; joints [-33.055, 44.931, -67.083, 35.093, 108.423, 12.52]
  Call Extruder(433.20001)
  MoveL 520 to (241.11, 53.34, 22.22) mm, rotated rx -180 ry 0 rz -180 deg; joints [-33.331, 44.964, -67.08, 35.371, 108.334, 12.588]
  MoveL 521 to (241.11, 53.34, 22.22) mm, rotated rx -180 ry 0 rz -180 deg; joints [-33.331, 44.964, -67.08, 35.371, 108.334, 12.588]
  Call Extruder(433.80182)
  MoveL 522 to (241.16, 53.93, 22.22) mm, rotated rx 180 ry 0 rz 180 deg; joints [-33.606, 44.997, -67.077, 35.646, 108.245, 12.654]
  MoveL 523 to (241.16, 53.93, 22.22) mm, rotated rx 180 ry 0 rz 180 deg; joints [-33.606, 44.997, -67.077, 35.646, 108.245, 12.654]
  Call Extruder(434.40048)
  MoveL 524 to (241.2, 54.52, 22.22) mm, rotated rx -180 ry 0 rz 180 deg; joints [-33.878, 45.03, -67.074, 35.919, 108.155, 12.719]
  MoveL 525 to (241.2, 54.52, 22.22) mm, rotated rx -180 ry 0 rz 180 deg; joints [-33.878, 45.03, -67.074, 35.919, 108.155, 12.719]
  Call Extruder(435.57226)
  MoveL 526 to (241.25, 55.68, 22.22) mm, rotated rx -180 ry 0 rz 180 deg; joints [-34.425, 45.092, -67.067, 36.466, 107.979, 12.85]
  MoveL 527 to (241.25, 55.68, 22.22) mm, rotated rx -180 ry 0 rz 180 deg; joints [-34.425, 45.092, -67.067, 36.466, 107.979, 12.85]
  Call Extruder(437.02987)
  MoveL 528 to (241.29, 57.14, 22.22) mm, rotated rx -180 ry 0 rz 180 deg; joints [-35.104, 45.17, -67.059, 37.145, 107.758, 13.01]
  Call Extruder(522.92352)
  MoveL 529 to (241.29, 142.86, 22.22) mm, rotated rx 180 ry 0 rz 180 deg; joints [-60.361, 50.533, -65.634, 61.218, 97.403, 13.199]
  Call Extruder(523.79834)
  MoveL 530 to (241.27, 143.73, 22.23) mm, rotated rx -180 ry 0 rz 180 deg; joints [-60.516, 50.588, -65.608, 61.361, 97.328, 13.147]
  MoveL 531 to (241.27, 143.73, 22.23) mm, rotated rx -180 ry 0 rz 180 deg; joints [-60.516, 50.588, -65.608, 61.361, 97.328, 13.147]
  Call Extruder(524.97012)
  MoveL 532 to (241.22, 144.9, 22.23) mm, rotated rx 180 ry 0 rz 180 deg; joints [-60.726, 50.662, -65.573, 61.556, 97.229, 13.077]
  MoveL 533 to (241.22, 144.9, 22.23) mm, rotated rx 180 ry 0 rz 180 deg; joints [-60.726, 50.662, -65.573, 61.556, 97.229, 13.077]
  Call Extruder(525.85826)
  MoveL 534 to (241.18, 145.77, 22.22) mm, rotated rx 180 ry 0 rz 180 deg; joints [-60.887, 50.717, -65.547, 61.705, 97.154, 13.025]
  MoveL 535 to (241.18, 145.77, 22.22) mm, rotated rx 180 ry 0 rz 180 deg; joints [-60.887, 50.717, -65.547, 61.705, 97.154, 13.025]
  Call Extruder(526.46008)
  MoveL 536 to (241.13, 146.36, 22.22) mm, rotated rx -180 ry 0 rz 180 deg; joints [-61, 50.753, -65.529, 61.809, 97.103, 12.991]
  MoveL 537 to (241.13, 146.36, 22.22) mm, rotated rx -180 ry 0 rz 180 deg; joints [-61, 50.753, -65.529, 61.809, 97.103, 12.991]
  Call Extruder(527.06505)
  MoveL 538 to (241.09, 146.95, 22.22) mm, rotated rx -180 ry 0 rz 180 deg; joints [-61.111, 50.789, -65.512, 61.913, 97.052, 12.956]
  MoveL 539 to (241.09, 146.95, 22.22) mm, rotated rx -180 ry 0 rz 180 deg; joints [-61.111, 50.789, -65.512, 61.913, 97.052, 12.956]
  Call Extruder(527.56965)
  MoveL 540 to (241.04, 147.44, 22.22) mm, rotated rx -180 ry 0 rz 180 deg; joints [-61.205, 50.819, -65.497, 62, 97.011, 12.928]
  MoveL 541 to (241.04, 147.44, 22.22) mm, rotated rx -180 ry 0 rz 180 deg; joints [-61.205, 50.819, -65.497, 62, 97.011, 12.928]
  Call Extruder(527.97299)
  MoveL 542 to (240.99, 147.83, 22.22) mm, rotated rx -180 ry 0 rz 180 deg; joints [-61.282, 50.842, -65.486, 62.072, 96.977, 12.907]
  MoveL 543 to (240.99, 147.83, 22.22) mm, rotated rx -180 ry 0 rz 180 deg; joints [-61.282, 50.842, -65.486, 62.072, 96.977, 12.907]
  Call Extruder(528.37839)
  MoveL 544 to (240.95, 148.22, 22.23) mm, rotated rx 180 ry 0 rz 180 deg; joints [-61.359, 50.865, -65.474, 62.144, 96.944, 12.885]
  MoveL 545 to (240.95, 148.22, 22.23) mm, rotated rx 180 ry 0 rz 180 deg; joints [-61.359, 50.865, -65.474, 62.144, 96.944, 12.885]
  Call Extruder(528.78583)
  MoveL 546 to (240.9, 148.6, 22.22) mm, rotated rx -180 ry 0 rz 180 deg; joints [-61.436, 50.889, -65.462, 62.215, 96.91, 12.863]
  MoveL 547 to (240.9, 148.6, 22.22) mm, rotated rx -180 ry 0 rz 180 deg; joints [-61.436, 50.889, -65.462, 62.215, 96.91, 12.863]
  Call Extruder(529.19532)
  MoveL 548 to (240.86, 148.99, 22.22) mm, rotated rx 180 ry 0 rz 180 deg; joints [-61.512, 50.912, -65.451, 62.287, 96.877, 12.841]
  MoveL 549 to (240.86, 148.99, 22.22) mm, rotated rx 180 ry 0 rz 180 deg; joints [-61.512, 50.912, -65.451, 62.287, 96.877, 12.841]
  Call Extruder(529.52188)
  MoveL 550 to (240.81, 149.3, 22.22) mm, rotated rx 180 ry 0 rz 180 deg; joints [-61.575, 50.93, -65.442, 62.346, 96.85, 12.824]
  MoveL 551 to (240.81, 149.3, 22.22) mm, rotated rx 180 ry 0 rz 180 deg; joints [-61.575, 50.93, -65.442, 62.346, 96.85, 12.824]
  Call Extruder(529.85015)
  MoveL 552 to (240.76, 149.6, 22.22) mm, rotated rx 180 ry 0 rz 180 deg; joints [-61.639, 50.948, -65.433, 62.406, 96.824, 12.807]
  MoveL 553 to (240.76, 149.6, 22.22) mm, rotated rx 180 ry 0 rz 180 deg; joints [-61.639, 50.948, -65.433, 62.406, 96.824, 12.807]
  Call Extruder(530.18015)
  MoveL 554 to (240.71, 149.91, 22.22) mm, rotated rx 180 ry 0 rz 180 deg; joints [-61.702, 50.966, -65.424, 62.465, 96.797, 12.791]
  MoveL 555 to (240.71, 149.91, 22.22) mm, rotated rx 180 ry 0 rz 180 deg; joints [-61.702, 50.966, -65.424, 62.465, 96.797, 12.791]
  Call Extruder(530.51186)
  MoveL 556 to (240.66, 150.21, 22.23) mm, rotated rx -180 ry 0 rz 180 deg; joints [-61.765, 50.984, -65.415, 62.524, 96.771, 12.774]
  MoveL 557 to (240.66, 150.21, 22.23) mm, rotated rx -180 ry 0 rz 180 deg; joints [-61.765, 50.984, -65.415, 62.524, 96.771, 12.774]
  Call Extruder(530.84529)
  MoveL 558 to (240.61, 150.52, 22.22) mm, rotated rx -180 ry 0 rz 180 deg; joints [-61.828, 51.002, -65.406, 62.583, 96.745, 12.757]
  MoveL 559 to (240.61, 150.52, 22.22) mm, rotated rx -180 ry 0 rz 180 deg; joints [-61.828, 51.002, -65.406, 62.583, 96.745, 12.757]
  Call Extruder(531.18045)
  MoveL 560 to (240.56, 150.83, 22.22) mm, rotated rx -180 ry 0 rz -180 deg; joints [-61.891, 51.02, -65.396, 62.642, 96.718, 12.74]
  MoveL 561 to (240.56, 150.83, 22.22) mm, rotated rx -180 ry 0 rz -180 deg; joints [-61.891, 51.02, -65.396, 62.642, 96.718, 12.74]
  Call Extruder(531.45690)
  MoveL 562 to (240.52, 151.07, 22.22) mm, rotated rx -180 ry 0 rz 180 deg; joints [-61.944, 51.034, -65.389, 62.692, 96.696, 12.727]
  MoveL 563 to (240.52, 151.07, 22.22) mm, rotated rx -180 ry 0 rz 180 deg; joints [-61.944, 51.034, -65.389, 62.692, 96.696, 12.727]
  Call Extruder(531.73480)
  MoveL 564 to (240.47, 151.32, 22.22) mm, rotated rx -180 ry 0 rz 180 deg; joints [-61.998, 51.048, -65.382, 62.743, 96.675, 12.714]
  MoveL 565 to (240.47, 151.32, 22.22) mm, rotated rx -180 ry 0 rz 180 deg; joints [-61.998, 51.048, -65.382, 62.743, 96.675, 12.714]
  Call Extruder(532.01414)
  MoveL 566 to (240.42, 151.57, 22.22) mm, rotated rx 180 ry 0 rz 180 deg; joints [-62.052, 51.062, -65.374, 62.793, 96.653, 12.7]
  MoveL 567 to (240.42, 151.57, 22.22) mm, rotated rx 180 ry 0 rz 180 deg; joints [-62.052, 51.062, -65.374, 62.793, 96.653, 12.7]
  Call Extruder(532.29492)
  MoveL 568 to (240.37, 151.82, 22.23) mm, rotated rx -180 ry 0 rz 180 deg; joints [-62.105, 51.077, -65.367, 62.844, 96.631, 12.687]
  MoveL 569 to (240.37, 151.82, 22.23) mm, rotated rx -180 ry 0 rz 180 deg; joints [-62.105, 51.077, -65.367, 62.844, 96.631, 12.687]
  Call Extruder(532.57714)
  MoveL 570 to (240.32, 152.07, 22.23) mm, rotated rx 180 ry 0 rz 180 deg; joints [-62.159, 51.091, -65.36, 62.894, 96.61, 12.674]
  MoveL 571 to (240.32, 152.07, 22.23) mm, rotated rx 180 ry 0 rz 180 deg; joints [-62.159, 51.091, -65.36, 62.894, 96.61, 12.674]
  Call Extruder(532.86081)
  MoveL 572 to (240.27, 152.32, 22.22) mm, rotated rx -180 ry 0 rz 180 deg; joints [-62.212, 51.105, -65.352, 62.944, 96.588, 12.66]
  MoveL 573 to (240.27, 152.32, 22.22) mm, rotated rx -180 ry 0 rz 180 deg; joints [-62.212, 51.105, -65.352, 62.944, 96.588, 12.66]
  Call Extruder(533.14591)
  MoveL 574 to (240.22, 152.57, 22.22) mm, rotated rx 180 ry 0 rz 180 deg; joints [-62.265, 51.119, -65.345, 62.994, 96.567, 12.647]
  MoveL 575 to (240.22, 152.57, 22.22) mm, rotated rx 180 ry 0 rz 180 deg; joints [-62.265, 51.119, -65.345, 62.994, 96.567, 12.647]
  Call Extruder(533.38165)
  MoveL 576 to (240.17, 152.77, 22.23) mm, rotated rx -180 ry 0 rz 180 deg; joints [-62.31, 51.131, -65.339, 63.036, 96.549, 12.636]
  MoveL 577 to (240.17, 152.77, 22.23) mm, rotated rx -180 ry 0 rz 180 deg; joints [-62.31, 51.131, -65.339, 63.036, 96.549, 12.636]
  Call Extruder(533.61845)
  MoveL 578 to (240.13, 152.98, 22.23) mm, rotated rx -180 ry 0 rz -180 deg; joints [-62.355, 51.143, -65.333, 63.078, 96.531, 12.625]
  MoveL 579 to (240.13, 152.98, 22.23) mm, rotated rx -180 ry 0 rz -180 deg; joints [-62.355, 51.143, -65.333, 63.078, 96.531, 12.625]
  Call Extruder(533.85633)
  MoveL 580 to (240.08, 153.18, 22.22) mm, rotated rx 180 ry 0 rz 180 deg; joints [-62.399, 51.154, -65.327, 63.12, 96.514, 12.614]
  MoveL 581 to (240.08, 153.18, 22.22) mm, rotated rx 180 ry 0 rz 180 deg; joints [-62.399, 51.154, -65.327, 63.12, 96.514, 12.614]
  Call Extruder(534.09527)
  MoveL 582 to (240.04, 153.39, 22.22) mm, rotated rx -180 ry 0 rz -180 deg; joints [-62.444, 51.166, -65.321, 63.162, 96.496, 12.604]
  MoveL 583 to (240.04, 153.39, 22.22) mm, rotated rx -180 ry 0 rz -180 deg; joints [-62.444, 51.166, -65.321, 63.162, 96.496, 12.604]
  Call Extruder(534.34924)
  MoveL 584 to (239.98, 153.6, 22.22) mm, rotated rx 180 ry 0 rz 180 deg; joints [-62.493, 51.178, -65.314, 63.208, 96.477, 12.593]
  MoveL 585 to (239.98, 153.6, 22.22) mm, rotated rx 180 ry 0 rz 180 deg; joints [-62.493, 51.178, -65.314, 63.208, 96.477, 12.593]
  Call Extruder(534.61883)
  MoveL 586 to (239.92, 153.82, 22.22) mm, rotated rx 180 ry 0 rz 180 deg; joints [-62.547, 51.19, -65.308, 63.259, 96.457, 12.582]
  MoveL 587 to (239.92, 153.82, 22.22) mm, rotated rx 180 ry 0 rz 180 deg; joints [-62.547, 51.19, -65.308, 63.259, 96.457, 12.582]
  Call Extruder(534.88976)
  MoveL 588 to (239.85, 154.05, 22.23) mm, rotated rx -180 ry 0 rz 180 deg; joints [-62.601, 51.202, -65.302, 63.31, 96.437, 12.572]
  MoveL 589 to (239.85, 154.05, 22.23) mm, rotated rx -180 ry 0 rz 180 deg; joints [-62.601, 51.202, -65.302, 63.31, 96.437, 12.572]
  Call Extruder(535.16202)
  MoveL 590 to (239.78, 154.27, 22.23) mm, rotated rx 180 ry 0 rz 180 deg; joints [-62.654, 51.214, -65.295, 63.361, 96.417, 12.561]
  MoveL 591 to (239.78, 154.27, 22.23) mm, rotated rx 180 ry 0 rz 180 deg; joints [-62.654, 51.214, -65.295, 63.361, 96.417, 12.561]
  Call Extruder(535.43561)
  MoveL 592 to (239.71, 154.49, 22.22) mm, rotated rx 180 ry 0 rz 180 deg; joints [-62.708, 51.226, -65.289, 63.412, 96.397, 12.55]
  MoveL 593 to (239.71, 154.49, 22.22) mm, rotated rx 180 ry 0 rz 180 deg; joints [-62.708, 51.226, -65.289, 63.412, 96.397, 12.55]
  Call Extruder(535.66881)
  MoveL 594 to (239.65, 154.68, 22.22) mm, rotated rx -180 ry 0 rz 180 deg; joints [-62.754, 51.236, -65.284, 63.456, 96.38, 12.541]
  MoveL 595 to (239.65, 154.68, 22.22) mm, rotated rx -180 ry 0 rz 180 deg; joints [-62.754, 51.236, -65.284, 63.456, 96.38, 12.541]
  Call Extruder(535.90306)
  MoveL 596 to (239.59, 154.87, 22.22) mm, rotated rx 180 ry 0 rz 180 deg; joints [-62.801, 51.246, -65.278, 63.5, 96.363, 12.533]
  MoveL 597 to (239.59, 154.87, 22.22) mm, rotated rx 180 ry 0 rz 180 deg; joints [-62.801, 51.246, -65.278, 63.5, 96.363, 12.533]
  Call Extruder(536.13835)
  MoveL 598 to (239.53, 155.06, 22.22) mm, rotated rx -180 ry 0 rz 180 deg; joints [-62.847, 51.256, -65.273, 63.544, 96.346, 12.524]
  MoveL 599 to (239.53, 155.06, 22.22) mm, rotated rx -180 ry 0 rz 180 deg; joints [-62.847, 51.256, -65.273, 63.544, 96.346, 12.524]
  Call Extruder(536.37470)
  MoveL 600 to (239.47, 155.25, 22.23) mm, rotated rx 180 ry 0 rz 180 deg; joints [-62.893, 51.266, -65.267, 63.588, 96.329, 12.515]
  MoveL 601 to (239.47, 155.25, 22.23) mm, rotated rx 180 ry 0 rz 180 deg; joints [-62.893, 51.266, -65.267, 63.588, 96.329, 12.515]
  Call Extruder(536.61210)
  MoveL 602 to (239.41, 155.44, 22.22) mm, rotated rx 180 ry 0 rz 180 deg; joints [-62.939, 51.276, -65.262, 63.632, 96.313, 12.506]
  MoveL 603 to (239.41, 155.44, 22.22) mm, rotated rx 180 ry 0 rz 180 deg; joints [-62.939, 51.276, -65.262, 63.632, 96.313, 12.506]
  Call Extruder(536.99230)
  MoveL 604 to (239.29, 155.73, 22.22) mm, rotated rx 180 ry 0 rz 180 deg; joints [-63.018, 51.291, -65.254, 63.707, 96.285, 12.494]
  MoveL 605 to (239.29, 155.73, 22.22) mm, rotated rx 180 ry 0 rz 180 deg; joints [-63.018, 51.291, -65.254, 63.707, 96.285, 12.494]
  Call Extruder(537.37429)
  MoveL 606 to (239.17, 156.02, 22.22) mm, rotated rx 180 ry 0 rz 180 deg; joints [-63.097, 51.305, -65.246, 63.782, 96.258, 12.482]
  MoveL 607 to (239.17, 156.02, 22.22) mm, rotated rx 180 ry 0 rz 180 deg; joints [-63.097, 51.305, -65.246, 63.782, 96.258, 12.482]
  Call Extruder(537.73076)
  MoveL 608 to (239.05, 156.29, 22.22) mm, rotated rx -180 ry 0 rz 180 deg; joints [-63.17, 51.319, -65.239, 63.852, 96.233, 12.471]
  MoveL 609 to (239.05, 156.29, 22.22) mm, rotated rx -180 ry 0 rz 180 deg; joints [-63.17, 51.319, -65.239, 63.852, 96.233, 12.471]
  Call Extruder(538.06143)
  MoveL 610 to (238.94, 156.54, 22.23) mm, rotated rx 180 ry 0 rz 180 deg; joints [-63.238, 51.331, -65.232, 63.917, 96.21, 12.461]
  MoveL 611 to (238.94, 156.54, 22.23) mm, rotated rx 180 ry 0 rz 180 deg; joints [-63.238, 51.331, -65.232, 63.917, 96.21, 12.461]
  Call Extruder(538.39353)
  MoveL 612 to (238.84, 156.79, 22.22) mm, rotated rx -180 ry 0 rz 180 deg; joints [-63.306, 51.344, -65.225, 63.981, 96.187, 12.451]
  MoveL 613 to (238.84, 156.79, 22.22) mm, rotated rx -180 ry 0 rz 180 deg; joints [-63.306, 51.344, -65.225, 63.981, 96.187, 12.451]
  Call Extruder(538.82540)
  MoveL 614 to (238.66, 157.09, 22.22) mm, rotated rx -180 ry 0 rz -180 deg; joints [-63.401, 51.358, -65.218, 64.073, 96.157, 12.442]
  MoveL 615 to (238.66, 157.09, 22.22) mm, rotated rx -180 ry 0 rz -180 deg; joints [-63.401, 51.358, -65.218, 64.073, 96.157, 12.442]
  Call Extruder(539.25912)
  MoveL 616 to (238.49, 157.4, 22.22) mm, rotated rx -180 ry 0 rz 180 deg; joints [-63.497, 51.371, -65.21, 64.165, 96.127, 12.432]
  MoveL 617 to (238.49, 157.4, 22.22) mm, rotated rx -180 ry 0 rz 180 deg; joints [-63.497, 51.371, -65.21, 64.165, 96.127, 12.432]
  Call Extruder(539.69468)
  MoveL 618 to (238.31, 157.7, 22.22) mm, rotated rx -180 ry 0 rz 180 deg; joints [-63.592, 51.385, -65.203, 64.256, 96.098, 12.423]
  MoveL 619 to (238.31, 157.7, 22.22) mm, rotated rx -180 ry 0 rz 180 deg; joints [-63.592, 51.385, -65.203, 64.256, 96.098, 12.423]
  Call Extruder(540.13207)
  MoveL 620 to (238.13, 158.01, 22.22) mm, rotated rx -180 ry 0 rz -180 deg; joints [-63.687, 51.399, -65.195, 64.348, 96.068, 12.413]
  MoveL 621 to (238.13, 158.01, 22.22) mm, rotated rx -180 ry 0 rz -180 deg; joints [-63.687, 51.399, -65.195, 64.348, 96.068, 12.413]
  Call Extruder(540.50882)
  MoveL 622 to (237.96, 158.25, 22.22) mm, rotated rx 180 ry 0 rz 180 deg; joints [-63.774, 51.409, -65.189, 64.431, 96.042, 12.408]
  MoveL 623 to (237.96, 158.25, 22.22) mm, rotated rx 180 ry 0 rz 180 deg; joints [-63.774, 51.409, -65.189, 64.431, 96.042, 12.408]
  Call Extruder(541.20873)
  MoveL 624 to (237.63, 158.7, 22.22) mm, rotated rx 180 ry 0 rz 180 deg; joints [-63.934, 51.428, -65.179, 64.586, 95.996, 12.398]
  MoveL 625 to (237.63, 158.7, 22.22) mm, rotated rx 180 ry 0 rz 180 deg; joints [-63.934, 51.428, -65.179, 64.586, 95.996, 12.398]
  Call Extruder(541.91145)
  MoveL 626 to (237.3, 159.15, 22.23) mm, rotated rx 180 ry 0 rz 180 deg; joints [-64.094, 51.446, -65.169, 64.74, 95.949, 12.388]
  Call Extruder(543.65031)
  MoveL 627 to (236.39, 160.19, 22.22) mm, rotated rx 180 ry 0 rz -180 deg; joints [-64.505, 51.485, -65.148, 65.138, 95.836, 12.376]
  Call Extruder(545.38913)
  MoveL 628 to (235.35, 161.1, 22.22) mm, rotated rx -180 ry 0 rz -180 deg; joints [-64.933, 51.512, -65.132, 65.554, 95.726, 12.379]
  Call Extruder(545.74051)
  MoveL 629 to (235.13, 161.27, 22.22) mm, rotated rx -180 ry 0 rz 180 deg; joints [-65.021, 51.515, -65.13, 65.64, 95.705, 12.383]
  MoveL 630 to (235.13, 161.27, 22.22) mm, rotated rx -180 ry 0 rz 180 deg; joints [-65.021, 51.515, -65.13, 65.64, 95.705, 12.383]
  Call Extruder(546.44047)
  MoveL 631 to (234.68, 161.6, 22.22) mm, rotated rx 180 ry 0 rz 180 deg; joints [-65.197, 51.523, -65.126, 65.812, 95.662, 12.389]
  MoveL 632 to (234.68, 161.6, 22.22) mm, rotated rx 180 ry 0 rz 180 deg; joints [-65.197, 51.523, -65.126, 65.812, 95.662, 12.389]
  Call Extruder(547.13763)
  MoveL 633 to (234.22, 161.92, 22.22) mm, rotated rx -180 ry 0 rz 180 deg; joints [-65.374, 51.531, -65.122, 65.984, 95.619, 12.395]
  MoveL 634 to (234.22, 161.92, 22.22) mm, rotated rx -180 ry 0 rz 180 deg; joints [-65.374, 51.531, -65.122, 65.984, 95.619, 12.395]
  Call Extruder(547.38444)
  MoveL 635 to (234.05, 162.02, 22.23) mm, rotated rx -180 ry 0 rz 180 deg; joints [-65.437, 51.532, -65.121, 66.046, 95.605, 12.399]
  MoveL 636 to (234.05, 162.02, 22.23) mm, rotated rx -180 ry 0 rz 180 deg; joints [-65.437, 51.532, -65.121, 66.046, 95.605, 12.399]
  Call Extruder(547.82000)
  MoveL 637 to (233.75, 162.2, 22.22) mm, rotated rx 180 ry 0 rz -180 deg; joints [-65.549, 51.535, -65.119, 66.156, 95.579, 12.406]
  MoveL 638 to (233.75, 162.2, 22.22) mm, rotated rx 180 ry 0 rz -180 deg; joints [-65.549, 51.535, -65.119, 66.156, 95.579, 12.406]
  Call Extruder(548.25372)
  MoveL 639 to (233.45, 162.37, 22.22) mm, rotated rx 180 ry 0 rz 180 deg; joints [-65.662, 51.537, -65.118, 66.266, 95.554, 12.413]
  MoveL 640 to (233.45, 162.37, 22.22) mm, rotated rx 180 ry 0 rz 180 deg; joints [-65.662, 51.537, -65.118, 66.266, 95.554, 12.413]
  Call Extruder(548.68559)
  MoveL 641 to (233.14, 162.55, 22.23) mm, rotated rx -180 ry 0 rz -180 deg; joints [-65.774, 51.539, -65.117, 66.376, 95.528, 12.42]
  MoveL 642 to (233.14, 162.55, 22.23) mm, rotated rx -180 ry 0 rz -180 deg; joints [-65.774, 51.539, -65.117, 66.376, 95.528, 12.42]
  Call Extruder(549.06597)
  MoveL 643 to (232.86, 162.69, 22.22) mm, rotated rx -180 ry 0 rz 180 deg; joints [-65.874, 51.541, -65.116, 66.474, 95.506, 12.428]
  MoveL 644 to (232.86, 162.69, 22.22) mm, rotated rx -180 ry 0 rz 180 deg; joints [-65.874, 51.541, -65.116, 66.474, 95.506, 12.428]
  Call Extruder(549.39656)
  MoveL 645 to (232.62, 162.8, 22.22) mm, rotated rx 180 ry 0 rz 180 deg; joints [-65.961, 51.54, -65.116, 66.559, 95.487, 12.437]
  MoveL 646 to (232.62, 162.8, 22.22) mm, rotated rx 180 ry 0 rz 180 deg; joints [-65.961, 51.54, -65.116, 66.559, 95.487, 12.437]
  Call Extruder(549.72573)
